LIN {X 0,Y 308.465,Z 992.055,A -85,B 0,C 180,E1 8309.518,E2 8309.518} C_VEL
LIN {X 0,Y 302.888,Z 996.087,A -85,B 0,C 180,E1 8308.383,E2 8308.383} C_VEL
LIN {X 0,Y 297.097,Z 1000.732,A -85,B 0,C 180,E1 8307.239,E2 8307.239} C_VEL
LIN {X 0,Y 292.705,Z 1003.413,A -85,B 0,C 180,E1 8306.146,E2 8306.146} C_VEL
LIN {X 0,Y 288.012,Z 1006.83,A -85,B 0,C 180,E1 8305.058,E2 8305.058} C_VEL
LIN {X 0,Y 284.129,Z 1009.021,A -85,B 0,C 180,E1 8303.872,E2 8303.872} C_VEL
LIN {X 0,Y 279.973,Z 1011.868,A -85,B 0,C 180,E1 8302.688,E2 8302.688} C_VEL
LIN {X 0,Y 277.713,Z 1012.755,A -85,B 0,C 180,E1 8301.768,E2 8301.768} C_VEL
LIN {X 0,Y 274.229,Z 1015.152,A -85,B 0,C 180,E1 8300.712,E2 8300.712} C_VEL
LIN {X 0,Y 271.961,Z 1016.233,A -85,B 0,C 180,E1 8299.546,E2 8299.546} C_VEL
LIN {X 0,Y 271.367,Z 1019.443,A -85,B 0,C 180,E1 8298.697,E2 8298.697} C_VEL
LIN {X 0,Y 269.802,Z 1031.042,A -85,B 0,C 180,E1 8295.696,E2 8295.696} C_VEL
LIN {X 0,Y 268.586,Z 1041.049,A -85,B 0,C 180,E1 8292.47,E2 8292.47} C_VEL
LIN {X 0,Y 267.824,Z 1048.97,A -85,B 0,C 180,E1 8289.238,E2 8289.238} C_VEL
LIN {X 0,Y 267.45,Z 1055.351,A -85,B 0,C 180,E1 8285.794,E2 8285.794} C_VEL
LIN {X 0,Y 267.481,Z 1059.896,A -85,B 0,C 180,E1 8282.357,E2 8282.357} C_VEL
LIN {X 0,Y 267.867,Z 1062.688,A -85,B 0,C 180,E1 8278.931,E2 8278.931} C_VEL
LIN {X 0,Y 268.592,Z 1063.764,A -85,B 0,C 180,E1 8275.517,E2 8275.517} C_VEL
LIN {X 0,Y 269.756,Z 1063.163,A -85,B 0,C 180,E1 8272.118,E2 8272.118} C_VEL
LIN {X 0,Y 271.423,Z 1060.847,A -85,B 0,C 180,E1 8268.742,E2 8268.742} C_VEL
LIN {X 0,Y 273.467,Z 1056.96,A -85,B 0,C 180,E1 8265.605,E2 8265.605} C_VEL
LIN {X 0,Y 276.201,Z 1050.914,A -85,B 0,C 180,E1 8262.298,E2 8262.298} C_VEL
LIN {X 0,Y 279.28,Z 1043.229,A -85,B 0,C 180,E1 8259.242,E2 8259.242} C_VEL
LIN {X 0,Y 282.707,Z 1033.633,A -85,B 0,C 180,E1 8256.351,E2 8256.351} C_VEL
LIN {X 0,Y 285.415,Z 1026.001,A -85,B 0,C 180,E1 8254.421,E2 8254.421} C_VEL
LIN {X 0,Y 288.972,Z 1024.505,A -85,B 0,C 180,E1 8253.491,E2 8253.491} C_VEL
LIN {X 0,Y 291.755,Z 1023.074,A -85,B 0,C 180,E1 8252.884,E2 8252.884} C_VEL
LIN {X 0,Y 296.745,Z 1020.577,A -85,B 0,C 180,E1 8251.855,E2 8251.855} C_VEL
LIN {X 0,Y 303.495,Z 1016.999,A -85,B 0,C 180,E1 8250.602,E2 8250.602} C_VEL
LIN {X 0,Y 312.335,Z 1011.631,A -85,B 0,C 180,E1 8249.19,E2 8249.19} C_VEL
LIN {X 0,Y 321.708,Z 1005.383,A -85,B 0,C 180,E1 8247.896,E2 8247.896} C_VEL
LIN {X 0,Y 326.811,Z 1001.618,A -85,B 0,C 180,E1 8247.283,E2 8247.283} C_VEL
LIN {X 0,Y 332.766,Z 996.983,A -85,B 0,C 180,E1 8246.592,E2 8246.592} C_VEL
LIN {X 0,Y 325.704,Z 1016.942,A -85,B 0,C 180,E1 8244.744,E2 8244.744} C_VEL
LIN {X 0,Y 318.629,Z 1034.815,A -85,B 0,C 180,E1 8242.726,E2 8242.726} C_VEL
LIN {X 0,Y 310.317,Z 1054.234,A -85,B 0,C 180,E1 8240.072,E2 8240.072} C_VEL
LIN {X 0,Y 302.689,Z 1070.961,A -85,B 0,C 180,E1 8237.305,E2 8237.305} C_VEL
LIN {X 0,Y 294.934,Z 1087.108,A -85,B 0,C 180,E1 8234.053,E2 8234.053} C_VEL
LIN {X 0,Y 287.656,Z 1102.055,A -85,B 0,C 180,E1 8230.429,E2 8230.429} C_VEL
LIN {X 0,Y 281.386,Z 1114.908,A -85,B 0,C 180,E1 8226.653,E2 8226.653} C_VEL
LIN {X 0,Y 275.565,Z 1127.286,A -85,B 0,C 180,E1 8222.234,E2 8222.234} C_VEL
LIN {X 0,Y 271.069,Z 1137.736,A -85,B 0,C 180,E1 8217.695,E2 8217.695} C_VEL
LIN {X 0,Y 267.812,Z 1146.209,A -85,B 0,C 180,E1 8213.08,E2 8213.08} C_VEL
LIN {X 0,Y 265.626,Z 1153.374,A -85,B 0,C 180,E1 8208.206,E2 8208.206} C_VEL
LIN {X 0,Y 264.507,Z 1158.372,A -85,B 0,C 180,E1 8203.719,E2 8203.719} C_VEL
LIN {X 0,Y 264.05,Z 1162.21,A -85,B 0,C 180,E1 8198.931,E2 8198.931} C_VEL
LIN {X 0,Y 263.973,Z 1164.181,A -85,B 0,C 180,E1 8194.78,E2 8194.78} C_VEL
LIN {X 0,Y 263.978,Z 1164.983,A -85,B 0,C 180,E1 8190.868,E2 8190.868} C_VEL
LIN {X 0,Y 263.962,Z 1164.612,A -85,B 0,C 180,E1 8186.525,E2 8186.525} C_VEL
LIN {X 0,Y 263.986,Z 1162.932,A -85,B 0,C 180,E1 8182.382,E2 8182.382} C_VEL
LIN {X 0,Y 264.232,Z 1160.273,A -85,B 0,C 180,E1 8178.431,E2 8178.431} C_VEL
LIN {X 0,Y 265.089,Z 1155.51,A -85,B 0,C 180,E1 8173.568,E2 8173.568} C_VEL
LIN {X 0,Y 266.681,Z 1149.663,A -85,B 0,C 180,E1 8169.134,E2 8169.134} C_VEL
LIN {X 0,Y 269.694,Z 1141.104,A -85,B 0,C 180,E1 8164.057,E2 8164.057} C_VEL
LIN {X 0,Y 273.705,Z 1131.511,A -85,B 0,C 180,E1 8159.484,E2 8159.484} C_VEL
LIN {X 0,Y 278.726,Z 1120.423,A -85,B 0,C 180,E1 8155.224,E2 8155.224} C_VEL
LIN {X 0,Y 284.969,Z 1107.485,A -85,B 0,C 180,E1 8151.093,E2 8151.093} C_VEL
LIN {X 0,Y 291.692,Z 1093.705,A -85,B 0,C 180,E1 8147.473,E2 8147.473} C_VEL
LIN {X 0,Y 299.455,Z 1077.629,A -85,B 0,C 180,E1 8143.986,E2 8143.986} C_VEL
LIN {X 0,Y 307.272,Z 1060.949,A -85,B 0,C 180,E1 8140.981,E2 8140.981} C_VEL
LIN {X 0,Y 315.017,Z 1043.264,A -85,B 0,C 180,E1 8138.374,E2 8138.374} C_VEL
LIN {X 0,Y 323.045,Z 1023.596,A -85,B 0,C 180,E1 8135.98,E2 8135.98} C_VEL
LIN {X 0,Y 330.114,Z 1004.598,A -85,B 0,C 180,E1 8134.078,E2 8134.078} C_VEL
LIN {X 0,Y 336.583,Z 984.934,A -85,B 0,C 180,E1 8132.472,E2 8132.472} C_VEL
LIN {X 0,Y 342.744,Z 963.75,A -85,B 0,C 180,E1 8131.059,E2 8131.059} C_VEL
LIN {X 0,Y 347.877,Z 942.3,A -85,B 0,C 180,E1 8129.938,E2 8129.938} C_VEL
LIN {X 0,Y 352.415,Z 919.016,A -85,B 0,C 180,E1 8129.004,E2 8129.004} C_VEL
LIN {X 0,Y 355.597,Z 897.104,A -85,B 0,C 180,E1 8128.357,E2 8128.357} C_VEL
LIN {X 0,Y 358.517,Z 862.586,A -85,B 0,C 180,E1 8127.602,E2 8127.602} C_VEL
LIN {X 0,Y 372.306,Z 678.191,A -85,B 0,C 180,E1 8123.839,E2 8123.839} C_VEL
LIN {X 0,Y 365.076,Z 666.2,A -85,B 0,C 180,E1 8120.857,E2 8120.857} C_VEL
LIN {X 0,Y 358.906,Z 656.732,A -85,B 0,C 180,E1 8117.928,E2 8117.928} C_VEL
LIN {X 0,Y 354.027,Z 649.555,A -85,B 0,C 180,E1 8115.227,E2 8115.227} C_VEL
LIN {X 0,Y 350.238,Z 644.346,A -85,B 0,C 180,E1 8112.782,E2 8112.782} C_VEL
LIN {X 0,Y 347.182,Z 640.185,A -85,B 0,C 180,E1 8110.453,E2 8110.453} C_VEL
LIN {X 0,Y 343.492,Z 635.283,A -85,B 0,C 180,E1 8106.854,E2 8106.854} C_VEL
LIN {X 0,Y 339.862,Z 631.157,A -85,B 0,C 180,E1 8100.505,E2 8100.505} C_VEL
LIN {X 0,Y 339.408,Z 630.8,A -85,B 0,C 180,E1 8097.467,E2 8097.467} C_VEL
LIN {X 0,Y 339.995,Z 632.727,A -85,B 0,C 180,E1 8093.414,E2 8093.414} C_VEL
LIN {X 0,Y 341.873,Z 635.288,A -85,B 0,C 180,E1 8089.808,E2 8089.808} C_VEL
LIN {X 0,Y 345.158,Z 640.526,A -85,B 0,C 180,E1 8085.916,E2 8085.916} C_VEL
LIN {X 0,Y 348.455,Z 645.83,A -85,B 0,C 180,E1 8083.067,E2 8083.067} C_VEL
LIN {X 0,Y 351.262,Z 650.243,A -85,B 0,C 180,E1 8081.064,E2 8081.064} C_VEL
LIN {X 0,Y 355.585,Z 657.064,A -85,B 0,C 180,E1 8078.429,E2 8078.429} C_VEL
LIN {X 0,Y 361.502,Z 667.073,A -85,B 0,C 180,E1 8075.357,E2 8075.357} C_VEL
LIN {X 0,Y 367.869,Z 678.378,A -85,B 0,C 180,E1 8072.524,E2 8072.524} C_VEL
LIN {X 0,Y 370.099,Z 682.724,A -85,B 0,C 180,E1 8071.607,E2 8071.607} C_VEL
LIN {X 0,Y 355.361,Z 895.308,A -85,B 0,C 180,E1 8067.466,E2 8067.466} C_VEL
LIN {X 0,Y 352.442,Z 917.469,A -85,B 0,C 180,E1 8066.87,E2 8066.87} C_VEL
LIN {X 0,Y 348.535,Z 938.899,A -85,B 0,C 180,E1 8066.077,E2 8066.077} C_VEL
LIN {X 0,Y 344.048,Z 958.089,A -85,B 0,C 180,E1 8065.133,E2 8065.133} C_VEL
LIN {X 0,Y 338.162,Z 979.093,A -85,B 0,C 180,E1 8063.823,E2 8063.823} C_VEL
LIN {X 0,Y 332.048,Z 997.764,A -85,B 0,C 180,E1 8062.368,E2 8062.368} C_VEL
LIN {X 0,Y 324.986,Z 1016.544,A -85,B 0,C 180,E1 8060.555,E2 8060.555} C_VEL
LIN {X 0,Y 317.727,Z 1034.044,A -85,B 0,C 180,E1 8058.501,E2 8058.501} C_VEL
LIN {X 0,Y 310.143,Z 1050.573,A -85,B 0,C 180,E1 8056.121,E2 8056.121} C_VEL
LIN {X 0,Y 302.083,Z 1066.923,A -85,B 0,C 180,E1 8053.247,E2 8053.247} C_VEL
LIN {X 0,Y 294.604,Z 1081.378,A -85,B 0,C 180,E1 8050.154,E2 8050.154} C_VEL
LIN {X 0,Y 287.561,Z 1094.347,A -85,B 0,C 180,E1 8046.731,E2 8046.731} C_VEL
LIN {X 0,Y 280.871,Z 1106.615,A -85,B 0,C 180,E1 8042.758,E2 8042.758} C_VEL
LIN {X 0,Y 275.408,Z 1116.941,A -85,B 0,C 180,E1 8038.635,E2 8038.635} C_VEL
LIN {X 0,Y 270.941,Z 1125.73,A -85,B 0,C 180,E1 8034.181,E2 8034.181} C_VEL
LIN {X 0,Y 267.62,Z 1133.095,A -85,B 0,C 180,E1 8029.421,E2 8029.421} C_VEL
LIN {X 0,Y 265.617,Z 1138.539,A -85,B 0,C 180,E1 8024.831,E2 8024.831} C_VEL
LIN {X 0,Y 264.545,Z 1142.323,A -85,B 0,C 180,E1 8020.232,E2 8020.232} C_VEL
LIN {X 0,Y 264.103,Z 1144.788,A -85,B 0,C 180,E1 8015.649,E2 8015.649} C_VEL
LIN {X 0,Y 264.011,Z 1145.742,A -85,B 0,C 180,E1 8011.302,E2 8011.302} C_VEL
LIN {X 0,Y 264.024,Z 1145.579,A -85,B 0,C 180,E1 8006.961,E2 8006.961} C_VEL
LIN {X 0,Y 264.22,Z 1143.987,A -85,B 0,C 180,E1 8002.509,E2 8002.509} C_VEL
LIN {X 0,Y 264.879,Z 1141.055,A -85,B 0,C 180,E1 7997.87,E2 7997.87} C_VEL
LIN {X 0,Y 266.314,Z 1136.484,A -85,B 0,C 180,E1 7993.196,E2 7993.196} C_VEL
LIN {X 0,Y 269.053,Z 1129.799,A -85,B 0,C 180,E1 7988.184,E2 7988.184} C_VEL
LIN {X 0,Y 272.827,Z 1121.996,A -85,B 0,C 180,E1 7983.676,E2 7983.676} C_VEL
LIN {X 0,Y 277.801,Z 1112.388,A -85,B 0,C 180,E1 7979.341,E2 7979.341} C_VEL
LIN {X 0,Y 283.954,Z 1101.024,A -85,B 0,C 180,E1 7975.219,E2 7975.219} C_VEL
LIN {X 0,Y 290.839,Z 1088.462,A -85,B 0,C 180,E1 7971.519,E2 7971.519} C_VEL
LIN {X 0,Y 297.873,Z 1075.192,A -85,B 0,C 180,E1 7968.347,E2 7968.347} C_VEL
LIN {X 0,Y 305.973,Z 1059.295,A -85,B 0,C 180,E1 7965.234,E2 7965.234} C_VEL
LIN {X 0,Y 310.204,Z 1050.584,A -85,B 0,C 180,E1 7963.776,E2 7963.776} C_VEL
LIN {X 0,Y 312.062,Z 1045.27,A -85,B 0,C 180,E1 7962.81,E2 7962.81} C_VEL
LIN {X 0,Y 314.292,Z 1031.888,A -85,B 0,C 180,E1 7960.095,E2 7960.095} C_VEL
LIN {X 0,Y 316.243,Z 1025.963,A -85,B 0,C 180,E1 7959.231,E2 7959.231} C_VEL
LIN {X 0,Y 324.268,Z 1006.326,A -85,B 0,C 180,E1 7957.149,E2 7957.149} C_VEL
LIN {X 0,Y 331.11,Z 987.486,A -85,B 0,C 180,E1 7955.529,E2 7955.529} C_VEL
LIN {X 0,Y 335.993,Z 971.645,A -85,B 0,C 180,E1 7954.403,E2 7954.403} C_VEL
LIN {X 0,Y 330.589,Z 977.083,A -85,B 0,C 180,E1 7953.722,E2 7953.722} C_VEL
LIN {X 0,Y 323.686,Z 984.266,A -85,B 0,C 180,E1 7952.934,E2 7952.934} C_VEL
LIN {X 0,Y 316.957,Z 990.052,A -85,B 0,C 180,E1 7951.942,E2 7951.942} C_VEL
LIN {X 0,Y 313.068,Z 993.358,A -85,B 0,C 180,E1 7951.372,E2 7951.372} C_VEL
LIN {X 0,Y 305.966,Z 999.179,A -85,B 0,C 180,E1 7950.216,E2 7950.216} C_VEL
LIN {X 0,Y 301.655,Z 1002.099,A -85,B 0,C 180,E1 7949.378,E2 7949.378} C_VEL
LIN {X 0,Y 295.641,Z 1006.57,A -85,B 0,C 180,E1 7948.261,E2 7948.261} C_VEL
LIN {X 0,Y 290.401,Z 1009.846,A -85,B 0,C 180,E1 7947.032,E2 7947.032} C_VEL
LIN {X 0,Y 285.061,Z 1013.4,A -85,B 0,C 180,E1 7945.782,E2 7945.782} C_VEL
LIN {X 0,Y 281.549,Z 1015.27,A -85,B 0,C 180,E1 7944.775,E2 7944.775} C_VEL
LIN {X 0,Y 276.925,Z 1018.136,A -85,B 0,C 180,E1 7943.495,E2 7943.495} C_VEL
LIN {X 0,Y 274.214,Z 1019.381,A -85,B 0,C 180,E1 7942.511,E2 7942.511} C_VEL
LIN {X 0,Y 270.333,Z 1021.776,A -85,B 0,C 180,E1 7941.252,E2 7941.252} C_VEL
LIN {X 0,Y 267.723,Z 1022.893,A -85,B 0,C 180,E1 7940.096,E2 7940.096} C_VEL
LIN {X 0,Y 264.674,Z 1024.759,A -85,B 0,C 180,E1 7938.959,E2 7938.959} C_VEL
LIN {X 0,Y 262.884,Z 1025.621,A -85,B 0,C 180,E1 7937.786,E2 7937.786} C_VEL
LIN {X 0,Y 261.135,Z 1038.389,A -85,B 0,C 180,E1 7933.959,E2 7933.959} C_VEL
LIN {X 0,Y 260.167,Z 1047.242,A -85,B 0,C 180,E1 7930.631,E2 7930.631} C_VEL
LIN {X 0,Y 259.621,Z 1054.468,A -85,B 0,C 180,E1 7927.08,E2 7927.08} C_VEL
LIN {X 0,Y 259.531,Z 1059.835,A -85,B 0,C 180,E1 7923.535,E2 7923.535} C_VEL
LIN {X 0,Y 259.82,Z 1063.351,A -85,B 0,C 180,E1 7920.001,E2 7920.001} C_VEL
LIN {X 0,Y 260.543,Z 1065.234,A -85,B 0,C 180,E1 7916.26,E2 7916.26} C_VEL
LIN {X 0,Y 261.684,Z 1065.286,A -85,B 0,C 180,E1 7912.757,E2 7912.757} C_VEL
LIN {X 0,Y 263.338,Z 1063.577,A -85,B 0,C 180,E1 7909.278,E2 7909.278} C_VEL
LIN {X 0,Y 265.727,Z 1059.828,A -85,B 0,C 180,E1 7905.621,E2 7905.621} C_VEL
LIN {X 0,Y 268.397,Z 1054.726,A -85,B 0,C 180,E1 7902.438,E2 7902.438} C_VEL
LIN {X 0,Y 271.579,Z 1047.72,A -85,B 0,C 180,E1 7899.303,E2 7899.303} C_VEL
LIN {X 0,Y 275.057,Z 1039.306,A -85,B 0,C 180,E1 7896.431,E2 7896.431} C_VEL
LIN {X 0,Y 277.235,Z 1034.271,A -85,B 0,C 180,E1 7894.928,E2 7894.928} C_VEL
LIN {X 0,Y 281.19,Z 1032.783,A -85,B 0,C 180,E1 7893.838,E2 7893.838} C_VEL
LIN {X 0,Y 287.246,Z 1030.196,A -85,B 0,C 180,E1 7892.423,E2 7892.423} C_VEL
LIN {X 0,Y 294.527,Z 1026.845,A -85,B 0,C 180,E1 7890.958,E2 7890.958} C_VEL
LIN {X 0,Y 302.933,Z 1022.356,A -85,B 0,C 180,E1 7889.481,E2 7889.481} C_VEL
LIN {X 0,Y 311.29,Z 1017.573,A -85,B 0,C 180,E1 7888.213,E2 7888.213} C_VEL
LIN {X 0,Y 321.765,Z 1010.786,A -85,B 0,C 180,E1 7886.846,E2 7886.846} C_VEL
LIN {X 0,Y 323.628,Z 1009.421,A -85,B 0,C 180,E1 7886.638,E2 7886.638} C_VEL
LIN {X 0,Y 315.936,Z 1029.029,A -85,B 0,C 180,E1 7884.58,E2 7884.58} C_VEL
LIN {X 0,Y 308.001,Z 1047.314,A -85,B 0,C 180,E1 7882.23,E2 7882.23} C_VEL
LIN {X 0,Y 299.535,Z 1065.454,A -85,B 0,C 180,E1 7879.39,E2 7879.39} C_VEL
LIN {X 0,Y 291.628,Z 1081.602,A -85,B 0,C 180,E1 7876.338,E2 7876.338} C_VEL
LIN {X 0,Y 283.839,Z 1096.749,A -85,B 0,C 180,E1 7872.834,E2 7872.834} C_VEL
LIN {X 0,Y 276.368,Z 1111.283,A -85,B 0,C 180,E1 7868.748,E2 7868.748} C_VEL
LIN {X 0,Y 270.14,Z 1123.702,A -85,B 0,C 180,E1 7864.492,E2 7864.492} C_VEL
LIN {X 0,Y 264.931,Z 1134.572,A -85,B 0,C 180,E1 7859.879,E2 7859.879} C_VEL
LIN {X 0,Y 260.916,Z 1144.044,A -85,B 0,C 180,E1 7854.932,E2 7854.932} C_VEL
LIN {X 0,Y 258.433,Z 1150.971,A -85,B 0,C 180,E1 7850.378,E2 7850.378} C_VEL
LIN {X 0,Y 256.814,Z 1156.919,A -85,B 0,C 180,E1 7845.352,E2 7845.352} C_VEL
LIN {X 0,Y 256.174,Z 1160.665,A -85,B 0,C 180,E1 7841.026,E2 7841.026} C_VEL
LIN {X 0,Y 255.982,Z 1163.366,A -85,B 0,C 180,E1 7836.504,E2 7836.504} C_VEL
LIN {X 0,Y 255.992,Z 1164.572,A -85,B 0,C 180,E1 7832.015,E2 7832.015} C_VEL
LIN {X 0,Y 255.993,Z 1164.595,A -85,B 0,C 180,E1 7828.209,E2 7828.209} C_VEL
LIN {X 0,Y 255.97,Z 1163.518,A -85,B 0,C 180,E1 7823.946,E2 7823.946} C_VEL
LIN {X 0,Y 256.127,Z 1160.994,A -85,B 0,C 180,E1 7819.428,E2 7819.428} C_VEL
LIN {X 0,Y 256.718,Z 1157.345,A -85,B 0,C 180,E1 7815.105,E2 7815.105} C_VEL
LIN {X 0,Y 258.237,Z 1151.588,A -85,B 0,C 180,E1 7810.079,E2 7810.079} C_VEL
LIN {X 0,Y 260.734,Z 1144.469,A -85,B 0,C 180,E1 7805.344,E2 7805.344} C_VEL
LIN {X 0,Y 264.764,Z 1134.908,A -85,B 0,C 180,E1 7800.292,E2 7800.292} C_VEL
LIN {X 0,Y 269.882,Z 1124.197,A -85,B 0,C 180,E1 7795.706,E2 7795.706} C_VEL
LIN {X 0,Y 276.016,Z 1111.888,A -85,B 0,C 180,E1 7791.46,E2 7791.46} C_VEL
LIN {X 0,Y 283.428,Z 1097.473,A -85,B 0,C 180,E1 7787.365,E2 7787.365} C_VEL
LIN {X 0,Y 290.827,Z 1083.025,A -85,B 0,C 180,E1 7783.984,E2 7783.984} C_VEL
LIN {X 0,Y 298.808,Z 1066.835,A -85,B 0,C 180,E1 7780.867,E2 7780.867} C_VEL
LIN {X 0,Y 306.909,Z 1049.674,A -85,B 0,C 180,E1 7778.115,E2 7778.115} C_VEL
LIN {X 0,Y 314.598,Z 1031.966,A -85,B 0,C 180,E1 7775.787,E2 7775.787} C_VEL
LIN {X 0,Y 322.793,Z 1011.438,A -85,B 0,C 180,E1 7773.567,E2 7773.567} C_VEL
LIN {X 0,Y 329.957,Z 991.415,A -85,B 0,C 180,E1 7771.805,E2 7771.805} C_VEL
LIN {X 0,Y 336.446,Z 970.408,A -85,B 0,C 180,E1 7770.326,E2 7770.326} C_VEL
LIN {X 0,Y 342.171,Z 948.852,A -85,B 0,C 180,E1 7769.107,E2 7769.107} C_VEL
LIN {X 0,Y 346.805,Z 927.205,A -85,B 0,C 180,E1 7768.161,E2 7768.161} C_VEL
LIN {X 0,Y 350.76,Z 903.276,A -85,B 0,C 180,E1 7767.394,E2 7767.394} C_VEL
LIN {X 0,Y 353.294,Z 879.798,A -85,B 0,C 180,E1 7766.833,E2 7766.833} C_VEL
LIN {X 0,Y 368.448,Z 682.805,A -85,B 0,C 180,E1 7762.812,E2 7762.812} C_VEL
LIN {X 0,Y 361.881,Z 671.774,A -85,B 0,C 180,E1 7759.951,E2 7759.951} C_VEL
LIN {X 0,Y 356.205,Z 662.826,A -85,B 0,C 180,E1 7757.099,E2 7757.099} C_VEL
LIN {X 0,Y 351.6,Z 656.045,A -85,B 0,C 180,E1 7754.408,E2 7754.408} C_VEL
LIN {X 0,Y 348.445,Z 651.582,A -85,B 0,C 180,E1 7752.259,E2 7752.259} C_VEL
LIN {X 0,Y 345.794,Z 647.871,A -85,B 0,C 180,E1 7750.159,E2 7750.159} C_VEL
LIN {X 0,Y 342.363,Z 643.155,A -85,B 0,C 180,E1 7746.708,E2 7746.708} C_VEL
LIN {X 0,Y 338.841,Z 639.045,A -85,B 0,C 180,E1 7740.338,E2 7740.338} C_VEL
LIN {X 0,Y 338.433,Z 638.746,A -85,B 0,C 180,E1 7737.46,E2 7737.46} C_VEL
LIN {X 0,Y 339.079,Z 640.829,A -85,B 0,C 180,E1 7733.226,E2 7733.226} C_VEL
LIN {X 0,Y 340.737,Z 643.111,A -85,B 0,C 180,E1 7730.03,E2 7730.03} C_VEL
LIN {X 0,Y 343.857,Z 648.243,A -85,B 0,C 180,E1 7726.205,E2 7726.205} C_VEL
LIN {X 0,Y 347.066,Z 653.562,A -85,B 0,C 180,E1 7723.342,E2 7723.342} C_VEL
LIN {X 0,Y 349.815,Z 658.024,A -85,B 0,C 180,E1 7721.329,E2 7721.329} C_VEL
LIN {X 0,Y 353.772,Z 664.454,A -85,B 0,C 180,E1 7718.842,E2 7718.842} C_VEL
LIN {X 0,Y 359.491,Z 674.372,A -85,B 0,C 180,E1 7715.779,E2 7715.779} C_VEL
LIN {X 0,Y 365.641,Z 685.618,A -85,B 0,C 180,E1 7712.959,E2 7712.959} C_VEL
LIN {X 0,Y 366.33,Z 687.354,A -85,B 0,C 180,E1 7712.647,E2 7712.647} C_VEL
LIN {X 0,Y 351.355,Z 895.604,A -85,B 0,C 180,E1 7708.589,E2 7708.589} C_VEL
LIN {X 0,Y 348.322,Z 917.825,A -85,B 0,C 180,E1 7707.991,E2 7707.991} C_VEL
LIN {X 0,Y 344.33,Z 939.046,A -85,B 0,C 180,E1 7707.209,E2 7707.209} C_VEL
LIN {X 0,Y 339.631,Z 958.56,A -85,B 0,C 180,E1 7706.252,E2 7706.252} C_VEL
LIN {X 0,Y 333.505,Z 979.699,A -85,B 0,C 180,E1 7704.931,E2 7704.931} C_VEL
LIN {X 0,Y 327.214,Z 998.316,A -85,B 0,C 180,E1 7703.48,E2 7703.48} C_VEL
LIN {X 0,Y 319.935,Z 1017.014,A -85,B 0,C 180,E1 7701.668,E2 7701.668} C_VEL
LIN {X 0,Y 312.275,Z 1034.784,A -85,B 0,C 180,E1 7699.567,E2 7699.567} C_VEL
LIN {X 0,Y 304.273,Z 1051.601,A -85,B 0,C 180,E1 7697.121,E2 7697.121} C_VEL
LIN {X 0,Y 296.085,Z 1067.512,A -85,B 0,C 180,E1 7694.282,E2 7694.282} C_VEL
LIN {X 0,Y 288.416,Z 1081.718,A -85,B 0,C 180,E1 7691.199,E2 7691.199} C_VEL
LIN {X 0,Y 281.047,Z 1094.68,A -85,B 0,C 180,E1 7687.728,E2 7687.728} C_VEL
LIN {X 0,Y 274.019,Z 1106.935,A -85,B 0,C 180,E1 7683.685,E2 7683.685} C_VEL
LIN {X 0,Y 268.244,Z 1117.252,A -85,B 0,C 180,E1 7679.474,E2 7679.474} C_VEL
LIN {X 0,Y 263.495,Z 1126.038,A -85,B 0,C 180,E1 7674.911,E2 7674.911} C_VEL
LIN {X 0,Y 259.939,Z 1133.397,A -85,B 0,C 180,E1 7670.02,E2 7670.02} C_VEL
LIN {X 0,Y 257.777,Z 1138.839,A -85,B 0,C 180,E1 7665.293,E2 7665.293} C_VEL
LIN {X 0,Y 256.598,Z 1142.619,A -85,B 0,C 180,E1 7660.553,E2 7660.553} C_VEL
LIN {X 0,Y 256.12,Z 1145.08,A -85,B 0,C 180,E1 7655.826,E2 7655.826} C_VEL
LIN {X 0,Y 256.014,Z 1146.011,A -85,B 0,C 180,E1 7651.567,E2 7651.567} C_VEL
LIN {X 0,Y 256.024,Z 1145.918,A -85,B 0,C 180,E1 7647.314,E2 7647.314} C_VEL
LIN {X 0,Y 256.223,Z 1144.434,A -85,B 0,C 180,E1 7642.601,E2 7642.601} C_VEL
LIN {X 0,Y 256.835,Z 1141.79,A -85,B 0,C 180,E1 7638.093,E2 7638.093} C_VEL
LIN {X 0,Y 258.339,Z 1137.265,A -85,B 0,C 180,E1 7633.125,E2 7633.125} C_VEL
LIN {X 0,Y 261.013,Z 1131.115,A -85,B 0,C 180,E1 7628.187,E2 7628.187} C_VEL
LIN {X 0,Y 264.847,Z 1123.5,A -85,B 0,C 180,E1 7623.546,E2 7623.546} C_VEL
LIN {X 0,Y 270.019,Z 1114.03,A -85,B 0,C 180,E1 7619.022,E2 7619.022} C_VEL
LIN {X 0,Y 276.233,Z 1103.191,A -85,B 0,C 180,E1 7614.864,E2 7614.864} C_VEL
LIN {X 0,Y 282.869,Z 1091.584,A -85,B 0,C 180,E1 7611.27,E2 7611.27} C_VEL
LIN {X 0,Y 290.474,Z 1078.009,A -85,B 0,C 180,E1 7607.838,E2 7607.838} C_VEL
LIN {X 0,Y 298.508,Z 1063.135,A -85,B 0,C 180,E1 7604.757,E2 7604.757} C_VEL
LIN {X 0,Y 306.418,Z 1047.36,A -85,B 0,C 180,E1 7602.114,E2 7602.114} C_VEL
LIN {X 0,Y 314.814,Z 1029.24,A -85,B 0,C 180,E1 7599.629,E2 7599.629} C_VEL
LIN {X 0,Y 316.243,Z 1025.963,A -85,B 0,C 180,E1 7599.231,E2 7599.231} C_VEL
LIN {X 0,Y 318.225,Z 1020.054,A -85,B 0,C 180,E1 7598.394,E2 7598.394} C_VEL
LIN {X 0,Y 320.783,Z 1005.274,A -85,B 0,C 180,E1 7595.988,E2 7595.988} C_VEL
LIN {X 0,Y 322.594,Z 998.896,A -85,B 0,C 180,E1 7595.275,E2 7595.275} C_VEL
LIN {X 0,Y 326.776,Z 987.099,A -85,B 0,C 180,E1 7594.296,E2 7594.296} C_VEL
LIN {X 0,Y 318.788,Z 994.051,A -85,B 0,C 180,E1 7593.29,E2 7593.29} C_VEL
LIN {X 0,Y 313.89,Z 997.958,A -85,B 0,C 180,E1 7592.57,E2 7592.57} C_VEL
LIN {X 0,Y 306.366,Z 1003.945,A -85,B 0,C 180,E1 7591.479,E2 7591.479} C_VEL
LIN {X 0,Y 299.562,Z 1008.615,A -85,B 0,C 180,E1 7590.265,E2 7590.265} C_VEL
LIN {X 0,Y 292.835,Z 1013.248,A -85,B 0,C 180,E1 7589.003,E2 7589.003} C_VEL
LIN {X 0,Y 288.024,Z 1016.094,A -85,B 0,C 180,E1 7587.947,E2 7587.947} C_VEL
LIN {X 0,Y 281.961,Z 1019.795,A -85,B 0,C 180,E1 7586.54,E2 7586.54} C_VEL
LIN {X 0,Y 278.95,Z 1021.394,A -85,B 0,C 180,E1 7585.704,E2 7585.704} C_VEL
LIN {X 0,Y 273.98,Z 1024.322,A -85,B 0,C 180,E1 7584.355,E2 7584.355} C_VEL
LIN {X 0,Y 270.732,Z 1025.831,A -85,B 0,C 180,E1 7583.277,E2 7583.277} C_VEL
LIN {X 0,Y 266.299,Z 1028.211,A -85,B 0,C 180,E1 7581.822,E2 7581.822} C_VEL
LIN {X 0,Y 263.979,Z 1029.196,A -85,B 0,C 180,E1 7580.858,E2 7580.858} C_VEL
LIN {X 0,Y 260.488,Z 1031.115,A -85,B 0,C 180,E1 7579.509,E2 7579.509} C_VEL
LIN {X 0,Y 258.622,Z 1031.734,A -85,B 0,C 180,E1 7578.483,E2 7578.483} C_VEL
LIN {X 0,Y 255.417,Z 1033.544,A -85,B 0,C 180,E1 7577.074,E2 7577.074} C_VEL
LIN {X 0,Y 253.98,Z 1034.217,A -85,B 0,C 180,E1 7575.912,E2 7575.912} C_VEL
LIN {X 0,Y 252.592,Z 1045.046,A -85,B 0,C 180,E1 7572.111,E2 7572.111} C_VEL
LIN {X 0,Y 251.846,Z 1053.216,A -85,B 0,C 180,E1 7568.448,E2 7568.448} C_VEL
LIN {X 0,Y 251.609,Z 1059.417,A -85,B 0,C 180,E1 7564.788,E2 7564.788} C_VEL
LIN {X 0,Y 251.793,Z 1063.683,A -85,B 0,C 180,E1 7561.138,E2 7561.138} C_VEL
LIN {X 0,Y 252.432,Z 1066.381,A -85,B 0,C 180,E1 7557.276,E2 7557.276} C_VEL
LIN {X 0,Y 253.508,Z 1067.185,A -85,B 0,C 180,E1 7553.66,E2 7553.66} C_VEL
LIN {X 0,Y 255.105,Z 1066.224,A -85,B 0,C 180,E1 7550.07,E2 7550.07} C_VEL
LIN {X 0,Y 257.318,Z 1063.568,A -85,B 0,C 180,E1 7546.519,E2 7546.519} C_VEL
LIN {X 0,Y 260.168,Z 1059.109,A -85,B 0,C 180,E1 7543.018,E2 7543.018} C_VEL
LIN {X 0,Y 263.627,Z 1052.577,A -85,B 0,C 180,E1 7539.579,E2 7539.579} C_VEL
LIN {X 0,Y 267.485,Z 1044.456,A -85,B 0,C 180,E1 7536.425,E2 7536.425} C_VEL
LIN {X 0,Y 268.698,Z 1042.164,A -85,B 0,C 180,E1 7535.604,E2 7535.604} C_VEL
LIN {X 0,Y 272.87,Z 1040.758,A -85,B 0,C 180,E1 7534.344,E2 7534.344} C_VEL
LIN {X 0,Y 278.591,Z 1038.738,A -85,B 0,C 180,E1 7532.882,E2 7532.882} C_VEL
LIN {X 0,Y 285.56,Z 1035.832,A -85,B 0,C 180,E1 7531.335,E2 7531.335} C_VEL
LIN {X 0,Y 292.991,Z 1032.477,A -85,B 0,C 180,E1 7529.891,E2 7529.891} C_VEL
LIN {X 0,Y 301.371,Z 1028.331,A -85,B 0,C 180,E1 7528.502,E2 7528.502} C_VEL
LIN {X 0,Y 311.108,Z 1022.839,A -85,B 0,C 180,E1 7527.103,E2 7527.103} C_VEL
LIN {X 0,Y 314.414,Z 1020.841,A -85,B 0,C 180,E1 7526.678,E2 7526.678} C_VEL
LIN {X 0,Y 306.51,Z 1039.334,A -85,B 0,C 180,E1 7524.505,E2 7524.505} C_VEL
LIN {X 0,Y 298.235,Z 1056.835,A -85,B 0,C 180,E1 7521.986,E2 7521.986} C_VEL
LIN {X 0,Y 289.319,Z 1074.577,A -85,B 0,C 180,E1 7518.885,E2 7518.885} C_VEL
LIN {X 0,Y 281.01,Z 1090.43,A -85,B 0,C 180,E1 7515.498,E2 7515.498} C_VEL
LIN {X 0,Y 273.115,Z 1104.93,A -85,B 0,C 180,E1 7511.684,E2 7511.684} C_VEL
LIN {X 0,Y 266.072,Z 1118.018,A -85,B 0,C 180,E1 7507.501,E2 7507.501} C_VEL
LIN {X 0,Y 260.2,Z 1129.246,A -85,B 0,C 180,E1 7503.104,E2 7503.104} C_VEL
LIN {X 0,Y 255.285,Z 1139.36,A -85,B 0,C 180,E1 7498.209,E2 7498.209} C_VEL
LIN {X 0,Y 251.887,Z 1147.439,A -85,B 0,C 180,E1 7493.388,E2 7493.388} C_VEL
LIN {X 0,Y 249.632,Z 1153.97,A -85,B 0,C 180,E1 7488.332,E2 7488.332} C_VEL
LIN {X 0,Y 248.43,Z 1159.005,A -85,B 0,C 180,E1 7483.262,E2 7483.262} C_VEL
LIN {X 0,Y 248.033,Z 1162.23,A -85,B 0,C 180,E1 7478.344,E2 7478.344} C_VEL
LIN {X 0,Y 247.978,Z 1163.961,A -85,B 0,C 180,E1 7473.93,E2 7473.93} C_VEL
LIN {X 0,Y 247.99,Z 1164.448,A -85,B 0,C 180,E1 7469.538,E2 7469.538} C_VEL
LIN {X 0,Y 247.98,Z 1163.739,A -85,B 0,C 180,E1 7465.375,E2 7465.375} C_VEL
LIN {X 0,Y 248.047,Z 1161.979,A -85,B 0,C 180,E1 7461.189,E2 7461.189} C_VEL
LIN {X 0,Y 248.537,Z 1158.358,A -85,B 0,C 180,E1 7456.032,E2 7456.032} C_VEL
LIN {X 0,Y 249.744,Z 1153.556,A -85,B 0,C 180,E1 7451.32,E2 7451.32} C_VEL
LIN {X 0,Y 252.162,Z 1146.671,A -85,B 0,C 180,E1 7446.144,E2 7446.144} C_VEL
LIN {X 0,Y 255.546,Z 1138.772,A -85,B 0,C 180,E1 7441.488,E2 7441.488} C_VEL
LIN {X 0,Y 260.693,Z 1128.205,A -85,B 0,C 180,E1 7436.475,E2 7436.475} C_VEL
LIN {X 0,Y 266.724,Z 1116.781,A -85,B 0,C 180,E1 7432.064,E2 7432.064} C_VEL
LIN {X 0,Y 273.641,Z 1103.891,A -85,B 0,C 180,E1 7428.036,E2 7428.036} C_VEL
LIN {X 0,Y 281.687,Z 1088.999,A -85,B 0,C 180,E1 7424.192,E2 7424.192} C_VEL
LIN {X 0,Y 289.812,Z 1073.532,A -85,B 0,C 180,E1 7420.926,E2 7420.926} C_VEL
LIN {X 0,Y 298.448,Z 1056.246,A -85,B 0,C 180,E1 7417.938,E2 7417.938} C_VEL
LIN {X 0,Y 306.739,Z 1038.646,A -85,B 0,C 180,E1 7415.421,E2 7415.421} C_VEL
LIN {X 0,Y 314.867,Z 1019.555,A -85,B 0,C 180,E1 7413.202,E2 7413.202} C_VEL
LIN {X 0,Y 323.109,Z 998.069,A -85,B 0,C 180,E1 7411.171,E2 7411.171} C_VEL
LIN {X 0,Y 330.062,Z 977.575,A -85,B 0,C 180,E1 7409.609,E2 7409.609} C_VEL
LIN {X 0,Y 336.184,Z 956.083,A -85,B 0,C 180,E1 7408.315,E2 7408.315} C_VEL
LIN {X 0,Y 341.658,Z 932.954,A -85,B 0,C 180,E1 7407.227,E2 7407.227} C_VEL
LIN {X 0,Y 345.704,Z 911.251,A -85,B 0,C 180,E1 7406.466,E2 7406.466} C_VEL
LIN {X 0,Y 348.707,Z 887.805,A -85,B 0,C 180,E1 7405.861,E2 7405.861} C_VEL
LIN {X 0,Y 364.554,Z 689.512,A -85,B 0,C 180,E1 7401.812,E2 7401.812} C_VEL
LIN {X 0,Y 364.617,Z 687.297,A -85,B 0,C 180,E1 7401.727,E2 7401.727} C_VEL
LIN {X 0,Y 358.248,Z 676.429,A -85,B 0,C 180,E1 7398.763,E2 7398.763} C_VEL
LIN {X 0,Y 352.499,Z 667.366,A -85,B 0,C 180,E1 7395.632,E2 7395.632} C_VEL
LIN {X 0,Y 347.775,Z 660.269,A -85,B 0,C 180,E1 7392.536,E2 7392.536} C_VEL
LIN {X 0,Y 344.417,Z 655.556,A -85,B 0,C 180,E1 7389.862,E2 7389.862} C_VEL
LIN {X 0,Y 341.097,Z 650.894,A -85,B 0,C 180,E1 7386.395,E2 7386.395} C_VEL
LIN {X 0,Y 337.823,Z 646.934,A -85,B 0,C 180,E1 7380.169,E2 7380.169} C_VEL
LIN {X 0,Y 337.455,Z 646.727,A -85,B 0,C 180,E1 7377.282,E2 7377.282} C_VEL
LIN {X 0,Y 338.377,Z 649.277,A -85,B 0,C 180,E1 7372.529,E2 7372.529} C_VEL
LIN {X 0,Y 339.654,Z 651.054,A -85,B 0,C 180,E1 7370.169,E2 7370.169} C_VEL
LIN {X 0,Y 342.562,Z 655.958,A -85,B 0,C 180,E1 7366.496,E2 7366.496} C_VEL
LIN {X 0,Y 345.686,Z 661.292,A -85,B 0,C 180,E1 7363.619,E2 7363.619} C_VEL
LIN {X 0,Y 348.258,Z 665.598,A -85,B 0,C 180,E1 7361.676,E2 7361.676} C_VEL
LIN {X 0,Y 352,Z 671.884,A -85,B 0,C 180,E1 7359.246,E2 7359.246} C_VEL
LIN {X 0,Y 357.657,Z 681.929,A -85,B 0,C 180,E1 7356.13,E2 7356.13} C_VEL
LIN {X 0,Y 362.706,Z 691.656,A -85,B 0,C 180,E1 7353.714,E2 7353.714} C_VEL
LIN {X 0,Y 347.518,Z 895.563,A -85,B 0,C 180,E1 7349.745,E2 7349.745} C_VEL
LIN {X 0,Y 344.4,Z 917.803,A -85,B 0,C 180,E1 7349.15,E2 7349.15} C_VEL
LIN {X 0,Y 340.262,Z 939.193,A -85,B 0,C 180,E1 7348.368,E2 7348.368} C_VEL
LIN {X 0,Y 335.344,Z 959.043,A -85,B 0,C 180,E1 7347.4,E2 7347.4} C_VEL
LIN {X 0,Y 328.976,Z 980.302,A -85,B 0,C 180,E1 7346.071,E2 7346.071} C_VEL
LIN {X 0,Y 322.19,Z 999.733,A -85,B 0,C 180,E1 7344.55,E2 7344.55} C_VEL
LIN {X 0,Y 314.673,Z 1018.27,A -85,B 0,C 180,E1 7342.732,E2 7342.732} C_VEL
LIN {X 0,Y 306.074,Z 1037.295,A -85,B 0,C 180,E1 7340.43,E2 7340.43} C_VEL
LIN {X 0,Y 297.739,Z 1054.15,A -85,B 0,C 180,E1 7337.916,E2 7337.916} C_VEL
LIN {X 0,Y 289.444,Z 1069.456,A -85,B 0,C 180,E1 7335.085,E2 7335.085} C_VEL
LIN {X 0,Y 280.966,Z 1084.306,A -85,B 0,C 180,E1 7331.718,E2 7331.718} C_VEL
LIN {X 0,Y 273.445,Z 1097.055,A -85,B 0,C 180,E1 7328.167,E2 7328.167} C_VEL
LIN {X 0,Y 266.57,Z 1108.363,A -85,B 0,C 180,E1 7324.238,E2 7324.238} C_VEL
LIN {X 0,Y 260.326,Z 1118.885,A -85,B 0,C 180,E1 7319.7,E2 7319.7} C_VEL
LIN {X 0,Y 255.492,Z 1127.512,A -85,B 0,C 180,E1 7315.002,E2 7315.002} C_VEL
LIN {X 0,Y 251.877,Z 1134.566,A -85,B 0,C 180,E1 7309.962,E2 7309.962} C_VEL
LIN {X 0,Y 249.547,Z 1140.122,A -85,B 0,C 180,E1 7304.621,E2 7304.621} C_VEL
LIN {X 0,Y 248.495,Z 1143.667,A -85,B 0,C 180,E1 7299.729,E2 7299.729} C_VEL
LIN {X 0,Y 248.083,Z 1145.688,A -85,B 0,C 180,E1 7294.855,E2 7294.855} C_VEL
LIN {X 0,Y 248.018,Z 1146.409,A -85,B 0,C 180,E1 7290.462,E2 7290.462} C_VEL
LIN {X 0,Y 248.064,Z 1145.91,A -85,B 0,C 180,E1 7285.839,E2 7285.839} C_VEL
LIN {X 0,Y 248.329,Z 1144.301,A -85,B 0,C 180,E1 7281.432,E2 7281.432} C_VEL
LIN {X 0,Y 249.258,Z 1140.996,A -85,B 0,C 180,E1 7276.31,E2 7276.31} C_VEL
LIN {X 0,Y 251.124,Z 1136.301,A -85,B 0,C 180,E1 7271.372,E2 7271.372} C_VEL
LIN {X 0,Y 254.289,Z 1129.729,A -85,B 0,C 180,E1 7266.355,E2 7266.355} C_VEL
LIN {X 0,Y 258.959,Z 1121.291,A -85,B 0,C 180,E1 7261.395,E2 7261.395} C_VEL
LIN {X 0,Y 264.545,Z 1111.857,A -85,B 0,C 180,E1 7257.026,E2 7257.026} C_VEL
LIN {X 0,Y 271.032,Z 1101.052,A -85,B 0,C 180,E1 7253.035,E2 7253.035} C_VEL
LIN {X 0,Y 278.647,Z 1088.387,A -85,B 0,C 180,E1 7249.227,E2 7249.227} C_VEL
LIN {X 0,Y 286.373,Z 1075.055,A -85,B 0,C 180,E1 7245.988,E2 7245.988} C_VEL
LIN {X 0,Y 294.922,Z 1059.539,A -85,B 0,C 180,E1 7242.921,E2 7242.921} C_VEL
LIN {X 0,Y 303.103,Z 1043.737,A -85,B 0,C 180,E1 7240.358,E2 7240.358} C_VEL
LIN {X 0,Y 311.204,Z 1026.386,A -85,B 0,C 180,E1 7238.079,E2 7238.079} C_VEL
LIN {X 0,Y 319.48,Z 1006.817,A -85,B 0,C 180,E1 7236,E2 7236} C_VEL
LIN {X 0,Y 322.594,Z 998.896,A -85,B 0,C 180,E1 7235.275,E2 7235.275} C_VEL
LIN {X 0,Y 322.388,Z 997.968,A -85,B 0,C 180,E1 7235.047,E2 7235.047} C_VEL
LIN {X 0,Y 320.677,Z 998.091,A -85,B 0,C 180,E1 7234.591,E2 7234.591} C_VEL
LIN {X 0,Y 317.5,Z 999.976,A -85,B 0,C 180,E1 7234.051,E2 7234.051} C_VEL
LIN {X 0,Y 307.008,Z 1008.567,A -85,B 0,C 180,E1 7232.752,E2 7232.752} C_VEL
LIN {X 0,Y 306.32,Z 1009.064,A -85,B 0,C 180,E1 7232.647,E2 7232.647} C_VEL
LIN {X 0,Y 298.265,Z 1014.392,A -85,B 0,C 180,E1 7231.306,E2 7231.306} C_VEL
LIN {X 0,Y 290.944,Z 1019.133,A -85,B 0,C 180,E1 7230,E2 7230} C_VEL
LIN {X 0,Y 286.41,Z 1021.747,A -85,B 0,C 180,E1 7229.029,E2 7229.029} C_VEL
LIN {X 0,Y 279.718,Z 1025.65,A -85,B 0,C 180,E1 7227.565,E2 7227.565} C_VEL
LIN {X 0,Y 275.569,Z 1027.799,A -85,B 0,C 180,E1 7226.506,E2 7226.506} C_VEL
LIN {X 0,Y 269.987,Z 1030.736,A -85,B 0,C 180,E1 7224.973,E2 7224.973} C_VEL
LIN {X 0,Y 267.163,Z 1032.089,A -85,B 0,C 180,E1 7224.076,E2 7224.076} C_VEL
LIN {X 0,Y 262.222,Z 1034.563,A -85,B 0,C 180,E1 7222.415,E2 7222.415} C_VEL
LIN {X 0,Y 260.239,Z 1035.412,A -85,B 0,C 180,E1 7221.645,E2 7221.645} C_VEL
LIN {X 0,Y 256.196,Z 1037.355,A -85,B 0,C 180,E1 7220.087,E2 7220.087} C_VEL
LIN {X 0,Y 254.097,Z 1038.146,A -85,B 0,C 180,E1 7219.063,E2 7219.063} C_VEL
LIN {X 0,Y 250.587,Z 1039.842,A -85,B 0,C 180,E1 7217.413,E2 7217.413} C_VEL
LIN {X 0,Y 249.26,Z 1040.227,A -85,B 0,C 180,E1 7216.522,E2 7216.522} C_VEL
LIN {X 0,Y 246.479,Z 1041.732,A -85,B 0,C 180,E1 7215.048,E2 7215.048} C_VEL
LIN {X 0,Y 245.182,Z 1042.286,A -85,B 0,C 180,E1 7213.802,E2 7213.802} C_VEL
LIN {X 0,Y 244.06,Z 1052.562,A -85,B 0,C 180,E1 7209.432,E2 7209.432} C_VEL
LIN {X 0,Y 243.697,Z 1059.31,A -85,B 0,C 180,E1 7205.652,E2 7205.652} C_VEL
LIN {X 0,Y 243.816,Z 1064.2,A -85,B 0,C 180,E1 7201.881,E2 7201.881} C_VEL
LIN {X 0,Y 244.378,Z 1067.359,A -85,B 0,C 180,E1 7198.125,E2 7198.125} C_VEL
LIN {X 0,Y 245.394,Z 1068.769,A -85,B 0,C 180,E1 7194.389,E2 7194.389} C_VEL
LIN {X 0,Y 247.093,Z 1068.435,A -85,B 0,C 180,E1 7190.451,E2 7190.451} C_VEL
LIN {X 0,Y 249.354,Z 1066.394,A -85,B 0,C 180,E1 7186.788,E2 7186.788} C_VEL
LIN {X 0,Y 252.272,Z 1062.501,A -85,B 0,C 180,E1 7183.183,E2 7183.183} C_VEL
LIN {X 0,Y 255.878,Z 1056.747,A -85,B 0,C 180,E1 7179.65,E2 7179.65} C_VEL
LIN {X 0,Y 260.153,Z 1049.471,A -85,B 0,C 180,E1 7176.321,E2 7176.321} C_VEL
LIN {X 0,Y 264.394,Z 1048.334,A -85,B 0,C 180,E1 7174.942,E2 7174.942} C_VEL
LIN {X 0,Y 269.942,Z 1046.617,A -85,B 0,C 180,E1 7173.374,E2 7173.374} C_VEL
LIN {X 0,Y 275.874,Z 1044.538,A -85,B 0,C 180,E1 7171.891,E2 7171.891} C_VEL
LIN {X 0,Y 283.065,Z 1041.736,A -85,B 0,C 180,E1 7170.363,E2 7170.363} C_VEL
LIN {X 0,Y 290.727,Z 1038.523,A -85,B 0,C 180,E1 7168.945,E2 7168.945} C_VEL
LIN {X 0,Y 300.518,Z 1033.711,A -85,B 0,C 180,E1 7167.386,E2 7167.386} C_VEL
LIN {X 0,Y 305.065,Z 1031.545,A -85,B 0,C 180,E1 7166.697,E2 7166.697} C_VEL
LIN {X 0,Y 296.347,Z 1050.184,A -85,B 0,C 180,E1 7164.237,E2 7164.237} C_VEL
LIN {X 0,Y 287.616,Z 1067.205,A -85,B 0,C 180,E1 7161.461,E2 7161.461} C_VEL
LIN {X 0,Y 278.329,Z 1084.377,A -85,B 0,C 180,E1 7158.041,E2 7158.041} C_VEL
LIN {X 0,Y 270.008,Z 1099.224,A -85,B 0,C 180,E1 7154.418,E2 7154.418} C_VEL
LIN {X 0,Y 262.334,Z 1112.587,A -85,B 0,C 180,E1 7150.387,E2 7150.387} C_VEL
LIN {X 0,Y 255.458,Z 1124.834,A -85,B 0,C 180,E1 7145.886,E2 7145.886} C_VEL
LIN {X 0,Y 250.054,Z 1134.891,A -85,B 0,C 180,E1 7141.32,E2 7141.32} C_VEL
LIN {X 0,Y 245.551,Z 1144.165,A -85,B 0,C 180,E1 7136.089,E2 7136.089} C_VEL
LIN {X 0,Y 242.644,Z 1151.313,A -85,B 0,C 180,E1 7131.008,E2 7131.008} C_VEL
LIN {X 0,Y 240.916,Z 1156.758,A -85,B 0,C 180,E1 7125.898,E2 7125.898} C_VEL
LIN {X 0,Y 240.196,Z 1160.412,A -85,B 0,C 180,E1 7121.283,E2 7121.283} C_VEL
LIN {X 0,Y 239.981,Z 1163.012,A -85,B 0,C 180,E1 7116.219,E2 7116.219} C_VEL
LIN {X 0,Y 240.002,Z 1164.015,A -85,B 0,C 180,E1 7111.91,E2 7111.91} C_VEL
LIN {X 0,Y 240.002,Z 1164.013,A -85,B 0,C 180,E1 7108.09,E2 7108.09} C_VEL
LIN {X 0,Y 239.987,Z 1162.933,A -85,B 0,C 180,E1 7103.541,E2 7103.541} C_VEL
LIN {X 0,Y 240.221,Z 1160.229,A -85,B 0,C 180,E1 7098.475,E2 7098.475} C_VEL
LIN {X 0,Y 240.974,Z 1156.523,A -85,B 0,C 180,E1 7093.859,E2 7093.859} C_VEL
LIN {X 0,Y 242.982,Z 1150.333,A -85,B 0,C 180,E1 7088.263,E2 7088.263} C_VEL
LIN {X 0,Y 246.08,Z 1143.022,A -85,B 0,C 180,E1 7083.191,E2 7083.191} C_VEL
LIN {X 0,Y 250.538,Z 1133.896,A -85,B 0,C 180,E1 7078.211,E2 7078.211} C_VEL
LIN {X 0,Y 256.35,Z 1123.208,A -85,B 0,C 180,E1 7073.462,E2 7073.462} C_VEL
LIN {X 0,Y 263.197,Z 1111.005,A -85,B 0,C 180,E1 7069.11,E2 7069.11} C_VEL
LIN {X 0,Y 271.314,Z 1096.763,A -85,B 0,C 180,E1 7064.962,E2 7064.962} C_VEL
LIN {X 0,Y 279.815,Z 1081.681,A -85,B 0,C 180,E1 7061.376,E2 7061.376} C_VEL
LIN {X 0,Y 288.412,Z 1065.532,A -85,B 0,C 180,E1 7058.258,E2 7058.258} C_VEL
LIN {X 0,Y 297.496,Z 1047.569,A -85,B 0,C 180,E1 7055.41,E2 7055.41} C_VEL
LIN {X 0,Y 305.867,Z 1029.601,A -85,B 0,C 180,E1 7053.086,E2 7053.086} C_VEL
LIN {X 0,Y 313.966,Z 1010.398,A -85,B 0,C 180,E1 7051.056,E2 7051.056} C_VEL
LIN {X 0,Y 321.635,Z 990.188,A -85,B 0,C 180,E1 7049.31,E2 7049.31} C_VEL
LIN {X 0,Y 328.165,Z 970.063,A -85,B 0,C 180,E1 7047.923,E2 7047.923} C_VEL
LIN {X 0,Y 334.349,Z 947.816,A -85,B 0,C 180,E1 7046.696,E2 7046.696} C_VEL
LIN {X 0,Y 339.139,Z 926.463,A -85,B 0,C 180,E1 7045.788,E2 7045.788} C_VEL
LIN {X 0,Y 343.162,Z 903.023,A -85,B 0,C 180,E1 7045.058,E2 7045.058} C_VEL
LIN {X 0,Y 345.813,Z 879.399,A -85,B 0,C 180,E1 7044.5,E2 7044.5} C_VEL
LIN {X 0,Y 361.075,Z 692.134,A -85,B 0,C 180,E1 7040.695,E2 7040.695} C_VEL
LIN {X 0,Y 355.12,Z 681.873,A -85,B 0,C 180,E1 7037.745,E2 7037.745} C_VEL
LIN {X 0,Y 350.304,Z 674.109,A -85,B 0,C 180,E1 7034.969,E2 7034.969} C_VEL
LIN {X 0,Y 345.78,Z 667.233,A -85,B 0,C 180,E1 7031.847,E2 7031.847} C_VEL
LIN {X 0,Y 343.056,Z 663.241,A -85,B 0,C 180,E1 7029.562,E2 7029.562} C_VEL
LIN {X 0,Y 339.961,Z 658.751,A -85,B 0,C 180,E1 7026.229,E2 7026.229} C_VEL
LIN {X 0,Y 336.805,Z 654.824,A -85,B 0,C 180,E1 7020,E2 7020} C_VEL
LIN {X 0,Y 336.48,Z 654.677,A -85,B 0,C 180,E1 7017.274,E2 7017.274} C_VEL
LIN {X 0,Y 337.729,Z 657.687,A -85,B 0,C 180,E1 7011.83,E2 7011.83} C_VEL
LIN {X 0,Y 338.574,Z 658.995,A -85,B 0,C 180,E1 7010.309,E2 7010.309} C_VEL
LIN {X 0,Y 341.272,Z 663.671,A -85,B 0,C 180,E1 7006.789,E2 7006.789} C_VEL
LIN {X 0,Y 344.219,Z 668.85,A -85,B 0,C 180,E1 7003.981,E2 7003.981} C_VEL
LIN {X 0,Y 346.936,Z 673.557,A -85,B 0,C 180,E1 7001.865,E2 7001.865} C_VEL
LIN {X 0,Y 350.428,Z 679.657,A -85,B 0,C 180,E1 6999.541,E2 6999.541} C_VEL
LIN {X 0,Y 355.682,Z 689.275,A -85,B 0,C 180,E1 6996.561,E2 6996.561} C_VEL
LIN {X 0,Y 359.183,Z 696.289,A -85,B 0,C 180,E1 6994.796,E2 6994.796} C_VEL
LIN {X 0,Y 343.83,Z 895.447,A -85,B 0,C 180,E1 6990.927,E2 6990.927} C_VEL
LIN {X 0,Y 340.63,Z 917.739,A -85,B 0,C 180,E1 6990.337,E2 6990.337} C_VEL
LIN {X 0,Y 336.337,Z 939.334,A -85,B 0,C 180,E1 6989.555,E2 6989.555} C_VEL
LIN {X 0,Y 331.427,Z 958.652,A -85,B 0,C 180,E1 6988.624,E2 6988.624} C_VEL
LIN {X 0,Y 324.92,Z 979.909,A -85,B 0,C 180,E1 6987.313,E2 6987.313} C_VEL
LIN {X 0,Y 317.93,Z 999.409,A -85,B 0,C 180,E1 6985.803,E2 6985.803} C_VEL
LIN {X 0,Y 310.21,Z 1017.945,A -85,B 0,C 180,E1 6984,E2 6984} C_VEL
LIN {X 0,Y 301.608,Z 1036.473,A -85,B 0,C 180,E1 6981.784,E2 6981.784} C_VEL
LIN {X 0,Y 293.216,Z 1052.902,A -85,B 0,C 180,E1 6979.359,E2 6979.359} C_VEL
LIN {X 0,Y 284.785,Z 1068.009,A -85,B 0,C 180,E1 6976.616,E2 6976.616} C_VEL
LIN {X 0,Y 276.344,Z 1082.393,A -85,B 0,C 180,E1 6973.429,E2 6973.429} C_VEL
LIN {X 0,Y 268.229,Z 1095.451,A -85,B 0,C 180,E1 6969.834,E2 6969.834} C_VEL
LIN {X 0,Y 260.546,Z 1107.573,A -85,B 0,C 180,E1 6965.684,E2 6965.684} C_VEL
LIN {X 0,Y 254.097,Z 1117.871,A -85,B 0,C 180,E1 6961.293,E2 6961.293} C_VEL
LIN {X 0,Y 248.736,Z 1126.654,A -85,B 0,C 180,E1 6956.5,E2 6956.5} C_VEL
LIN {X 0,Y 244.616,Z 1134.086,A -85,B 0,C 180,E1 6951.259,E2 6951.259} C_VEL
LIN {X 0,Y 242.05,Z 1139.638,A -85,B 0,C 180,E1 6946.067,E2 6946.067} C_VEL
LIN {X 0,Y 240.687,Z 1143.359,A -85,B 0,C 180,E1 6941.017,E2 6941.017} C_VEL
LIN {X 0,Y 240.143,Z 1145.726,A -85,B 0,C 180,E1 6935.975,E2 6935.975} C_VEL
LIN {X 0,Y 240.026,Z 1146.614,A -85,B 0,C 180,E1 6931.432,E2 6931.432} C_VEL
LIN {X 0,Y 240.042,Z 1146.479,A -85,B 0,C 180,E1 6926.896,E2 6926.896} C_VEL
LIN {X 0,Y 240.276,Z 1144.996,A -85,B 0,C 180,E1 6922.053,E2 6922.053} C_VEL
LIN {X 0,Y 241.079,Z 1142.237,A -85,B 0,C 180,E1 6917.073,E2 6917.073} C_VEL
LIN {X 0,Y 242.796,Z 1137.86,A -85,B 0,C 180,E1 6912.009,E2 6912.009} C_VEL
LIN {X 0,Y 245.911,Z 1131.715,A -85,B 0,C 180,E1 6906.767,E2 6906.767} C_VEL
LIN {X 0,Y 250.281,Z 1124.108,A -85,B 0,C 180,E1 6901.874,E2 6901.874} C_VEL
LIN {X 0,Y 256.099,Z 1114.652,A -85,B 0,C 180,E1 6897.133,E2 6897.133} C_VEL
LIN {X 0,Y 263.003,Z 1103.835,A -85,B 0,C 180,E1 6892.809,E2 6892.809} C_VEL
LIN {X 0,Y 270.304,Z 1092.235,A -85,B 0,C 180,E1 6889.101,E2 6889.101} C_VEL
LIN {X 0,Y 278.629,Z 1078.637,A -85,B 0,C 180,E1 6885.571,E2 6885.571} C_VEL
LIN {X 0,Y 287.297,Z 1063.861,A -85,B 0,C 180,E1 6882.455,E2 6882.455} C_VEL
LIN {X 0,Y 295.89,Z 1047.946,A -85,B 0,C 180,E1 6879.757,E2 6879.757} C_VEL
LIN {X 0,Y 305.069,Z 1029.439,A -85,B 0,C 180,E1 6877.209,E2 6877.209} C_VEL
LIN {X 0,Y 313.228,Z 1011.299,A -85,B 0,C 180,E1 6875.196,E2 6875.196} C_VEL
LIN {X 0,Y 317.551,Z 1000.459,A -85,B 0,C 180,E1 6874.166,E2 6874.166} C_VEL
LIN {X 0,Y 312.014,Z 1004.743,A -85,B 0,C 180,E1 6873.448,E2 6873.448} C_VEL
LIN {X 0,Y 306.32,Z 1009.064,A -85,B 0,C 180,E1 6872.647,E2 6872.647} C_VEL
LIN {X 0,Y 302.717,Z 1012.204,A -85,B 0,C 180,E1 6872.225,E2 6872.225} C_VEL
LIN {X 0,Y 293.397,Z 1021.846,A -85,B 0,C 180,E1 6871.636,E2 6871.636} C_VEL
LIN {X 0,Y 289.751,Z 1024.579,A -85,B 0,C 180,E1 6871.148,E2 6871.148} C_VEL
LIN {X 0,Y 283.185,Z 1028.211,A -85,B 0,C 180,E1 6869.858,E2 6869.858} C_VEL
LIN {X 0,Y 276.194,Z 1031.972,A -85,B 0,C 180,E1 6868.31,E2 6868.31} C_VEL
LIN {X 0,Y 267.083,Z 1036.571,A -85,B 0,C 180,E1 6865.977,E2 6865.977} C_VEL
LIN {X 0,Y 263.419,Z 1038.242,A -85,B 0,C 180,E1 6864.882,E2 6864.882} C_VEL
LIN {X 0,Y 257.93,Z 1040.693,A -85,B 0,C 180,E1 6863.05,E2 6863.05} C_VEL
LIN {X 0,Y 251.791,Z 1043.469,A -85,B 0,C 180,E1 6860.697,E2 6860.697} C_VEL
LIN {X 0,Y 249.491,Z 1044.417,A -85,B 0,C 180,E1 6859.645,E2 6859.645} C_VEL
LIN {X 0,Y 245.691,Z 1046.023,A -85,B 0,C 180,E1 6857.772,E2 6857.772} C_VEL
LIN {X 0,Y 244.121,Z 1046.649,A -85,B 0,C 180,E1 6856.906,E2 6856.906} C_VEL
LIN {X 0,Y 241.115,Z 1047.932,A -85,B 0,C 180,E1 6855.145,E2 6855.145} C_VEL
LIN {X 0,Y 239.964,Z 1048.272,A -85,B 0,C 180,E1 6854.232,E2 6854.232} C_VEL
LIN {X 0,Y 237.322,Z 1049.602,A -85,B 0,C 180,E1 6852.408,E2 6852.408} C_VEL
LIN {X 0,Y 236.458,Z 1050.212,A -85,B 0,C 180,E1 6851.161,E2 6851.161} C_VEL
LIN {X 0,Y 235.842,Z 1058.215,A -85,B 0,C 180,E1 6847.063,E2 6847.063} C_VEL
LIN {X 0,Y 235.809,Z 1063.922,A -85,B 0,C 180,E1 6843.16,E2 6843.16} C_VEL
LIN {X 0,Y 236.27,Z 1067.873,A -85,B 0,C 180,E1 6839.273,E2 6839.273} C_VEL
LIN {X 0,Y 237.193,Z 1070.055,A -85,B 0,C 180,E1 6835.407,E2 6835.407} C_VEL
LIN {X 0,Y 238.817,Z 1070.553,A -85,B 0,C 180,E1 6831.332,E2 6831.332} C_VEL
LIN {X 0,Y 241.032,Z 1069.319,A -85,B 0,C 180,E1 6827.544,E2 6827.544} C_VEL
LIN {X 0,Y 244.144,Z 1066.044,A -85,B 0,C 180,E1 6823.586,E2 6823.586} C_VEL
LIN {X 0,Y 247.841,Z 1061.129,A -85,B 0,C 180,E1 6819.946,E2 6819.946} C_VEL
LIN {X 0,Y 250.985,Z 1056.505,A -85,B 0,C 180,E1 6817.392,E2 6817.392} C_VEL
LIN {X 0,Y 255.454,Z 1055.511,A -85,B 0,C 180,E1 6815.735,E2 6815.735} C_VEL
LIN {X 0,Y 260.639,Z 1054.181,A -85,B 0,C 180,E1 6814.067,E2 6814.067} C_VEL
LIN {X 0,Y 271.013,Z 1051.119,A -85,B 0,C 180,E1 6811.341,E2 6811.341} C_VEL
LIN {X 0,Y 280.56,Z 1047.551,A -85,B 0,C 180,E1 6809.362,E2 6809.362} C_VEL
LIN {X 0,Y 289.615,Z 1043.759,A -85,B 0,C 180,E1 6807.762,E2 6807.762} C_VEL
LIN {X 0,Y 295.875,Z 1041.03,A -85,B 0,C 180,E1 6806.776,E2 6806.776} C_VEL
LIN {X 0,Y 287.535,Z 1057.46,A -85,B 0,C 180,E1 6804.372,E2 6804.372} C_VEL
LIN {X 0,Y 277.969,Z 1074.958,A -85,B 0,C 180,E1 6801.254,E2 6801.254} C_VEL
LIN {X 0,Y 269.286,Z 1090.103,A -85,B 0,C 180,E1 6797.954,E2 6797.954} C_VEL
LIN {X 0,Y 260.959,Z 1104,A -85,B 0,C 180,E1 6794.214,E2 6794.214} C_VEL
LIN {X 0,Y 253.239,Z 1116.873,A -85,B 0,C 180,E1 6790.008,E2 6790.008} C_VEL
LIN {X 0,Y 246.5,Z 1128.264,A -85,B 0,C 180,E1 6785.384,E2 6785.384} C_VEL
LIN {X 0,Y 240.759,Z 1138.601,A -85,B 0,C 180,E1 6780.166,E2 6780.166} C_VEL
LIN {X 0,Y 236.727,Z 1146.818,A -85,B 0,C 180,E1 6774.984,E2 6774.984} C_VEL
LIN {X 0,Y 234.065,Z 1153.236,A -85,B 0,C 180,E1 6769.723,E2 6769.723} C_VEL
LIN {X 0,Y 232.607,Z 1158.21,A -85,B 0,C 180,E1 6764.437,E2 6764.437} C_VEL
LIN {X 0,Y 232.064,Z 1161.52,A -85,B 0,C 180,E1 6759.173,E2 6759.173} C_VEL
LIN {X 0,Y 231.986,Z 1163.233,A -85,B 0,C 180,E1 6754.697,E2 6754.697} C_VEL
LIN {X 0,Y 232.013,Z 1163.908,A -85,B 0,C 180,E1 6750,E2 6750} C_VEL
LIN {X 0,Y 231.986,Z 1163.227,A -85,B 0,C 180,E1 6745.303,E2 6745.303} C_VEL
LIN {X 0,Y 232.064,Z 1161.51,A -85,B 0,C 180,E1 6740.827,E2 6740.827} C_VEL
LIN {X 0,Y 232.606,Z 1158.193,A -85,B 0,C 180,E1 6735.563,E2 6735.563} C_VEL
LIN {X 0,Y 233.973,Z 1153.484,A -85,B 0,C 180,E1 6730.529,E2 6730.529} C_VEL
LIN {X 0,Y 236.565,Z 1147.147,A -85,B 0,C 180,E1 6725.264,E2 6725.264} C_VEL
LIN {X 0,Y 240.53,Z 1138.988,A -85,B 0,C 180,E1 6720.077,E2 6720.077} C_VEL
LIN {X 0,Y 245.973,Z 1129.159,A -85,B 0,C 180,E1 6715.029,E2 6715.029} C_VEL
LIN {X 0,Y 252.197,Z 1118.5,A -85,B 0,C 180,E1 6710.629,E2 6710.629} C_VEL
LIN {X 0,Y 260.092,Z 1105.373,A -85,B 0,C 180,E1 6706.214,E2 6706.214} C_VEL
LIN {X 0,Y 268.455,Z 1091.401,A -85,B 0,C 180,E1 6702.386,E2 6702.386} C_VEL
LIN {X 0,Y 277.271,Z 1076.053,A -85,B 0,C 180,E1 6698.983,E2 6698.983} C_VEL
LIN {X 0,Y 286.5,Z 1059.308,A -85,B 0,C 180,E1 6695.937,E2 6695.937} C_VEL
LIN {X 0,Y 294.918,Z 1042.794,A -85,B 0,C 180,E1 6693.486,E2 6693.486} C_VEL
LIN {X 0,Y 304.292,Z 1022.764,A -85,B 0,C 180,E1 6691.056,E2 6691.056} C_VEL
LIN {X 0,Y 312.175,Z 1004.112,A -85,B 0,C 180,E1 6689.216,E2 6689.216} C_VEL
LIN {X 0,Y 319.675,Z 983.814,A -85,B 0,C 180,E1 6687.601,E2 6687.601} C_VEL
LIN {X 0,Y 326.224,Z 963.619,A -85,B 0,C 180,E1 6686.298,E2 6686.298} C_VEL
LIN {X 0,Y 331.866,Z 942.463,A -85,B 0,C 180,E1 6685.229,E2 6685.229} C_VEL
LIN {X 0,Y 336.806,Z 919.672,A -85,B 0,C 180,E1 6684.346,E2 6684.346} C_VEL
LIN {X 0,Y 340.276,Z 898.062,A -85,B 0,C 180,E1 6683.726,E2 6683.726} C_VEL
LIN {X 0,Y 343.451,Z 865.235,A -85,B 0,C 180,E1 6683.011,E2 6683.011} C_VEL
LIN {X 0,Y 357.564,Z 696.955,A -85,B 0,C 180,E1 6679.606,E2 6679.606} C_VEL
LIN {X 0,Y 352.175,Z 687.408,A -85,B 0,C 180,E1 6676.748,E2 6676.748} C_VEL
LIN {X 0,Y 347.331,Z 679.492,A -85,B 0,C 180,E1 6673.738,E2 6673.738} C_VEL
LIN {X 0,Y 343.74,Z 674.023,A -85,B 0,C 180,E1 6671.068,E2 6671.068} C_VEL
LIN {X 0,Y 341.612,Z 670.818,A -85,B 0,C 180,E1 6669.178,E2 6669.178} C_VEL
LIN {X 0,Y 338.723,Z 666.506,A -85,B 0,C 180,E1 6665.93,E2 6665.93} C_VEL
LIN {X 0,Y 335.787,Z 662.716,A -85,B 0,C 180,E1 6659.829,E2 6659.829} C_VEL
LIN {X 0,Y 335.503,Z 662.676,A -85,B 0,C 180,E1 6657.096,E2 6657.096} C_VEL
LIN {X 0,Y 337.273,Z 666.331,A -85,B 0,C 180,E1 6650.874,E2 6650.874} C_VEL
LIN {X 0,Y 339.99,Z 671.383,A -85,B 0,C 180,E1 6647.085,E2 6647.085} C_VEL
LIN {X 0,Y 342.855,Z 676.576,A -85,B 0,C 180,E1 6644.263,E2 6644.263} C_VEL
LIN {X 0,Y 346.541,Z 682.994,A -85,B 0,C 180,E1 6641.408,E2 6641.408} C_VEL
LIN {X 0,Y 351.968,Z 693.167,A -85,B 0,C 180,E1 6637.976,E2 6637.976} C_VEL
LIN {X 0,Y 355.793,Z 700.884,A -85,B 0,C 180,E1 6635.899,E2 6635.899} C_VEL
LIN {X 0,Y 340.283,Z 895.439,A -85,B 0,C 180,E1 6632.132,E2 6632.132} C_VEL
LIN {X 0,Y 337.006,Z 917.688,A -85,B 0,C 180,E1 6631.549,E2 6631.549} C_VEL
LIN {X 0,Y 332.559,Z 939.474,A -85,B 0,C 180,E1 6630.769,E2 6630.769} C_VEL
LIN {X 0,Y 327.349,Z 959.408,A -85,B 0,C 180,E1 6629.814,E2 6629.814} C_VEL
LIN {X 0,Y 320.672,Z 980.507,A -85,B 0,C 180,E1 6628.515,E2 6628.515} C_VEL
LIN {X 0,Y 313.491,Z 999.931,A -85,B 0,C 180,E1 6627.016,E2 6627.016} C_VEL
LIN {X 0,Y 305.549,Z 1018.408,A -85,B 0,C 180,E1 6625.221,E2 6625.221} C_VEL
LIN {X 0,Y 296.368,Z 1037.48,A -85,B 0,C 180,E1 6622.929,E2 6622.929} C_VEL
LIN {X 0,Y 287.409,Z 1054.393,A -85,B 0,C 180,E1 6620.405,E2 6620.405} C_VEL
LIN {X 0,Y 278.186,Z 1070.175,A -85,B 0,C 180,E1 6617.461,E2 6617.461} C_VEL
LIN {X 0,Y 269.003,Z 1084.981,A -85,B 0,C 180,E1 6614.032,E2 6614.032} C_VEL
LIN {X 0,Y 260.776,Z 1097.716,A -85,B 0,C 180,E1 6610.389,E2 6610.389} C_VEL
LIN {X 0,Y 253.194,Z 1109,A -85,B 0,C 180,E1 6606.324,E2 6606.324} C_VEL
LIN {X 0,Y 245.925,Z 1119.945,A -85,B 0,C 180,E1 6601.36,E2 6601.36} C_VEL
LIN {X 0,Y 240.529,Z 1128.488,A -85,B 0,C 180,E1 6596.41,E2 6596.41} C_VEL
LIN {X 0,Y 236.45,Z 1135.459,A -85,B 0,C 180,E1 6591.065,E2 6591.065} C_VEL
LIN {X 0,Y 233.875,Z 1140.716,A -85,B 0,C 180,E1 6585.625,E2 6585.625} C_VEL
LIN {X 0,Y 232.606,Z 1144.257,A -85,B 0,C 180,E1 6580.401,E2 6580.401} C_VEL
LIN {X 0,Y 232.118,Z 1146.208,A -85,B 0,C 180,E1 6575.438,E2 6575.438} C_VEL
LIN {X 0,Y 232.03,Z 1146.948,A -85,B 0,C 180,E1 6570.988,E2 6570.988} C_VEL
LIN {X 0,Y 232.07,Z 1146.62,A -85,B 0,C 180,E1 6566.047,E2 6566.047} C_VEL
LIN {X 0,Y 232.353,Z 1145.099,A -85,B 0,C 180,E1 6561.338,E2 6561.338} C_VEL
LIN {X 0,Y 233.318,Z 1142.175,A -85,B 0,C 180,E1 6556.114,E2 6556.114} C_VEL
LIN {X 0,Y 235.307,Z 1137.675,A -85,B 0,C 180,E1 6550.902,E2 6550.902} C_VEL
LIN {X 0,Y 239.061,Z 1130.879,A -85,B 0,C 180,E1 6545.175,E2 6545.175} C_VEL
LIN {X 0,Y 243.877,Z 1123.23,A -85,B 0,C 180,E1 6540.259,E2 6540.259} C_VEL
LIN {X 0,Y 250.257,Z 1113.47,A -85,B 0,C 180,E1 6535.435,E2 6535.435} C_VEL
LIN {X 0,Y 257.727,Z 1102.307,A -85,B 0,C 180,E1 6531.061,E2 6531.061} C_VEL
LIN {X 0,Y 266.019,Z 1089.806,A -85,B 0,C 180,E1 6527.132,E2 6527.132} C_VEL
LIN {X 0,Y 274.886,Z 1075.737,A -85,B 0,C 180,E1 6523.628,E2 6523.628} C_VEL
LIN {X 0,Y 284.309,Z 1059.909,A -85,B 0,C 180,E1 6520.455,E2 6520.455} C_VEL
LIN {X 0,Y 293.072,Z 1044.142,A -85,B 0,C 180,E1 6517.887,E2 6517.887} C_VEL
LIN {X 0,Y 301.841,Z 1026.578,A -85,B 0,C 180,E1 6515.587,E2 6515.587} C_VEL
LIN {X 0,Y 308.131,Z 1012.834,A -85,B 0,C 180,E1 6514.074,E2 6514.074} C_VEL
LIN {X 0,Y 299.438,Z 1018.391,A -85,B 0,C 180,E1 6512.748,E2 6512.748} C_VEL
LIN {X 0,Y 290.588,Z 1024.112,A -85,B 0,C 180,E1 6511.303,E2 6511.303} C_VEL
LIN {X 0,Y 289.751,Z 1024.579,A -85,B 0,C 180,E1 6511.148,E2 6511.148} C_VEL
LIN {X 0,Y 286.024,Z 1027.255,A -85,B 0,C 180,E1 6510.618,E2 6510.618} C_VEL
LIN {X 0,Y 276.224,Z 1035.896,A -85,B 0,C 180,E1 6509.73,E2 6509.73} C_VEL
LIN {X 0,Y 273.109,Z 1037.894,A -85,B 0,C 180,E1 6509.22,E2 6509.22} C_VEL
LIN {X 0,Y 272.641,Z 1038.109,A -85,B 0,C 180,E1 6509.108,E2 6509.108} C_VEL
LIN {X 0,Y 264.116,Z 1042.261,A -85,B 0,C 180,E1 6507.019,E2 6507.019} C_VEL
LIN {X 0,Y 254.624,Z 1046.419,A -85,B 0,C 180,E1 6504.104,E2 6504.104} C_VEL
LIN {X 0,Y 247.696,Z 1049.275,A -85,B 0,C 180,E1 6501.552,E2 6501.552} C_VEL
LIN {X 0,Y 244.838,Z 1050.396,A -85,B 0,C 180,E1 6500.312,E2 6500.312} C_VEL
LIN {X 0,Y 240.926,Z 1051.899,A -85,B 0,C 180,E1 6498.386,E2 6498.386} C_VEL
LIN {X 0,Y 236.231,Z 1053.809,A -85,B 0,C 180,E1 6495.717,E2 6495.717} C_VEL
LIN {X 0,Y 234.991,Z 1054.207,A -85,B 0,C 180,E1 6494.792,E2 6494.792} C_VEL
LIN {X 0,Y 232.065,Z 1055.541,A -85,B 0,C 180,E1 6492.694,E2 6492.694} C_VEL
LIN {X 0,Y 230.837,Z 1055.963,A -85,B 0,C 180,E1 6491.494,E2 6491.494} C_VEL
LIN {X 0,Y 228.535,Z 1057.101,A -85,B 0,C 180,E1 6489.317,E2 6489.317} C_VEL
LIN {X 0,Y 227.998,Z 1057.653,A -85,B 0,C 180,E1 6488.068,E2 6488.068} C_VEL
LIN {X 0,Y 227.857,Z 1063.991,A -85,B 0,C 180,E1 6484.027,E2 6484.027} C_VEL
LIN {X 0,Y 228.231,Z 1068.462,A -85,B 0,C 180,E1 6480.001,E2 6480.001} C_VEL
LIN {X 0,Y 229.208,Z 1071.371,A -85,B 0,C 180,E1 6475.748,E2 6475.748} C_VEL
LIN {X 0,Y 230.755,Z 1072.394,A -85,B 0,C 180,E1 6471.78,E2 6471.78} C_VEL
LIN {X 0,Y 232.984,Z 1071.682,A -85,B 0,C 180,E1 6467.862,E2 6467.862} C_VEL
LIN {X 0,Y 236.19,Z 1069.124,A -85,B 0,C 180,E1 6463.777,E2 6463.777} C_VEL
LIN {X 0,Y 240.011,Z 1064.926,A -85,B 0,C 180,E1 6460.026,E2 6460.026} C_VEL
LIN {X 0,Y 241.709,Z 1063.071,A -85,B 0,C 180,E1 6458.653,E2 6458.653} C_VEL
LIN {X 0,Y 249.708,Z 1061.692,A -85,B 0,C 180,E1 6455.392,E2 6455.392} C_VEL
LIN {X 0,Y 260.683,Z 1059.027,A -85,B 0,C 180,E1 6452.1,E2 6452.1} C_VEL
LIN {X 0,Y 274.091,Z 1054.708,A -85,B 0,C 180,E1 6449.046,E2 6449.046} C_VEL
LIN {X 0,Y 286.628,Z 1049.964,A -85,B 0,C 180,E1 6446.847,E2 6446.847} C_VEL
LIN {X 0,Y 276.928,Z 1067.48,A -85,B 0,C 180,E1 6443.975,E2 6443.975} C_VEL
LIN {X 0,Y 266.888,Z 1084.536,A -85,B 0,C 180,E1 6440.512,E2 6440.512} C_VEL
LIN {X 0,Y 257.81,Z 1099.316,A -85,B 0,C 180,E1 6436.813,E2 6436.813} C_VEL
LIN {X 0,Y 249.348,Z 1112.58,A -85,B 0,C 180,E1 6432.662,E2 6432.662} C_VEL
LIN {X 0,Y 241.246,Z 1125.442,A -85,B 0,C 180,E1 6427.665,E2 6427.665} C_VEL
LIN {X 0,Y 234.991,Z 1135.87,A -85,B 0,C 180,E1 6422.6,E2 6422.6} C_VEL
LIN {X 0,Y 230.109,Z 1144.657,A -85,B 0,C 180,E1 6417.145,E2 6417.145} C_VEL
LIN {X 0,Y 226.764,Z 1151.858,A -85,B 0,C 180,E1 6411.467,E2 6411.467} C_VEL
LIN {X 0,Y 224.976,Z 1156.816,A -85,B 0,C 180,E1 6406.26,E2 6406.26} C_VEL
LIN {X 0,Y 224.143,Z 1160.614,A -85,B 0,C 180,E1 6400.799,E2 6400.799} C_VEL
LIN {X 0,Y 223.98,Z 1162.648,A -85,B 0,C 180,E1 6395.893,E2 6395.893} C_VEL
LIN {X 0,Y 224.012,Z 1163.482,A -85,B 0,C 180,E1 6391.535,E2 6391.535} C_VEL
LIN {X 0,Y 223.99,Z 1163.356,A -85,B 0,C 180,E1 6387.186,E2 6387.186} C_VEL
LIN {X 0,Y 223.998,Z 1162.051,A -85,B 0,C 180,E1 6382.275,E2 6382.275} C_VEL
LIN {X 0,Y 224.365,Z 1159.293,A -85,B 0,C 180,E1 6377.125,E2 6377.125} C_VEL
LIN {X 0,Y 225.618,Z 1154.903,A -85,B 0,C 180,E1 6371.506,E2 6371.506} C_VEL
LIN {X 0,Y 228.078,Z 1148.759,A -85,B 0,C 180,E1 6365.94,E2 6365.94} C_VEL
LIN {X 0,Y 232.152,Z 1140.789,A -85,B 0,C 180,E1 6360.311,E2 6360.311} C_VEL
LIN {X 0,Y 237.313,Z 1131.823,A -85,B 0,C 180,E1 6355.334,E2 6355.334} C_VEL
LIN {X 0,Y 244.271,Z 1120.538,A -85,B 0,C 180,E1 6350.31,E2 6350.31} C_VEL
LIN {X 0,Y 252.322,Z 1107.912,A -85,B 0,C 180,E1 6345.779,E2 6345.779} C_VEL
LIN {X 0,Y 261.202,Z 1093.68,A -85,B 0,C 180,E1 6341.717,E2 6341.717} C_VEL
LIN {X 0,Y 271.217,Z 1077.162,A -85,B 0,C 180,E1 6337.915,E2 6337.915} C_VEL
LIN {X 0,Y 280.641,Z 1060.86,A -85,B 0,C 180,E1 6334.88,E2 6334.88} C_VEL
LIN {X 0,Y 289.777,Z 1043.614,A -85,B 0,C 180,E1 6332.289,E2 6332.289} C_VEL
LIN {X 0,Y 298.96,Z 1024.849,A -85,B 0,C 180,E1 6329.978,E2 6329.978} C_VEL
LIN {X 0,Y 306.707,Z 1007.2,A -85,B 0,C 180,E1 6328.209,E2 6328.209} C_VEL
LIN {X 0,Y 314.996,Z 985.919,A -85,B 0,C 180,E1 6326.475,E2 6326.475} C_VEL
LIN {X 0,Y 321.787,Z 965.74,A -85,B 0,C 180,E1 6325.161,E2 6325.161} C_VEL
LIN {X 0,Y 327.703,Z 944.609,A -85,B 0,C 180,E1 6324.077,E2 6324.077} C_VEL
LIN {X 0,Y 332.752,Z 922.684,A -85,B 0,C 180,E1 6323.205,E2 6323.205} C_VEL
LIN {X 0,Y 336.538,Z 900.189,A -85,B 0,C 180,E1 6322.553,E2 6322.553} C_VEL
LIN {X 0,Y 339.701,Z 869.886,A -85,B 0,C 180,E1 6321.884,E2 6321.884} C_VEL
LIN {X 0,Y 354.195,Z 701.749,A -85,B 0,C 180,E1 6318.495,E2 6318.495} C_VEL
LIN {X 0,Y 348.862,Z 692.339,A -85,B 0,C 180,E1 6315.458,E2 6315.458} C_VEL
LIN {X 0,Y 344.817,Z 685.632,A -85,B 0,C 180,E1 6312.731,E2 6312.731} C_VEL
LIN {X 0,Y 340.882,Z 679.24,A -85,B 0,C 180,E1 6309.454,E2 6309.454} C_VEL
LIN {X 0,Y 337.602,Z 674.377,A -85,B 0,C 180,E1 6305.779,E2 6305.779} C_VEL
LIN {X 0,Y 334.804,Z 670.668,A -85,B 0,C 180,E1 6299.828,E2 6299.828} C_VEL
LIN {X 0,Y 334.531,Z 670.631,A -85,B 0,C 180,E1 6297.087,E2 6297.087} C_VEL
LIN {X 0,Y 336.201,Z 674.273,A -85,B 0,C 180,E1 6291.017,E2 6291.017} C_VEL
LIN {X 0,Y 338.795,Z 679.249,A -85,B 0,C 180,E1 6287.298,E2 6287.298} C_VEL
LIN {X 0,Y 341.505,Z 684.301,A -85,B 0,C 180,E1 6284.548,E2 6284.548} C_VEL
LIN {X 0,Y 345.156,Z 690.928,A -85,B 0,C 180,E1 6281.637,E2 6281.637} C_VEL
LIN {X 0,Y 350.149,Z 700.621,A -85,B 0,C 180,E1 6278.385,E2 6278.385} C_VEL
LIN {X 0,Y 352.506,Z 705.745,A -85,B 0,C 180,E1 6277.019,E2 6277.019} C_VEL
LIN {X 0,Y 336.892,Z 895.383,A -85,B 0,C 180,E1 6273.362,E2 6273.362} C_VEL
LIN {X 0,Y 333.512,Z 917.766,A -85,B 0,C 180,E1 6272.783,E2 6272.783} C_VEL
LIN {X 0,Y 328.934,Z 939.609,A -85,B 0,C 180,E1 6272.011,E2 6272.011} C_VEL
LIN {X 0,Y 323.776,Z 958.888,A -85,B 0,C 180,E1 6271.103,E2 6271.103} C_VEL
LIN {X 0,Y 316.926,Z 980.109,A -85,B 0,C 180,E1 6269.818,E2 6269.818} C_VEL
LIN {X 0,Y 309.541,Z 999.604,A -85,B 0,C 180,E1 6268.336,E2 6268.336} C_VEL
LIN {X 0,Y 301.363,Z 1018.144,A -85,B 0,C 180,E1 6266.556,E2 6266.556} C_VEL
LIN {X 0,Y 292.207,Z 1036.689,A -85,B 0,C 180,E1 6264.358,E2 6264.358} C_VEL
LIN {X 0,Y 283.212,Z 1053.165,A -85,B 0,C 180,E1 6261.933,E2 6261.933} C_VEL
LIN {X 0,Y 273.866,Z 1068.723,A -85,B 0,C 180,E1 6259.09,E2 6259.09} C_VEL
LIN {X 0,Y 264.728,Z 1083.063,A -85,B 0,C 180,E1 6255.858,E2 6255.858} C_VEL
LIN {X 0,Y 255.957,Z 1096.004,A -85,B 0,C 180,E1 6252.214,E2 6252.214} C_VEL
LIN {X 0,Y 247.421,Z 1108.207,A -85,B 0,C 180,E1 6247.898,E2 6247.898} C_VEL
LIN {X 0,Y 240.238,Z 1118.486,A -85,B 0,C 180,E1 6243.324,E2 6243.324} C_VEL
LIN {X 0,Y 234.189,Z 1127.267,A -85,B 0,C 180,E1 6238.288,E2 6238.288} C_VEL
LIN {X 0,Y 229.515,Z 1134.603,A -85,B 0,C 180,E1 6232.813,E2 6232.813} C_VEL
LIN {X 0,Y 226.469,Z 1140.232,A -85,B 0,C 180,E1 6227.206,E2 6227.206} C_VEL
LIN {X 0,Y 224.845,Z 1143.95,A -85,B 0,C 180,E1 6221.804,E2 6221.804} C_VEL
LIN {X 0,Y 224.185,Z 1146.31,A -85,B 0,C 180,E1 6216.402,E2 6216.402} C_VEL
LIN {X 0,Y 224.036,Z 1147.196,A -85,B 0,C 180,E1 6211.534,E2 6211.534} C_VEL
LIN {X 0,Y 224.058,Z 1147.06,A -85,B 0,C 180,E1 6206.674,E2 6206.674} C_VEL
LIN {X 0,Y 224.337,Z 1145.605,A -85,B 0,C 180,E1 6201.542,E2 6201.542} C_VEL
LIN {X 0,Y 225.247,Z 1142.966,A -85,B 0,C 180,E1 6196.393,E2 6196.393} C_VEL
LIN {X 0,Y 227.354,Z 1138.455,A -85,B 0,C 180,E1 6190.741,E2 6190.741} C_VEL
LIN {X 0,Y 230.962,Z 1132.325,A -85,B 0,C 180,E1 6185.17,E2 6185.17} C_VEL
LIN {X 0,Y 235.948,Z 1124.714,A -85,B 0,C 180,E1 6179.997,E2 6179.997} C_VEL
LIN {X 0,Y 242.488,Z 1115.271,A -85,B 0,C 180,E1 6175.03,E2 6175.03} C_VEL
LIN {X 0,Y 250.151,Z 1104.474,A -85,B 0,C 180,E1 6170.541,E2 6170.541} C_VEL
LIN {X 0,Y 258.638,Z 1092.201,A -85,B 0,C 180,E1 6166.518,E2 6166.518} C_VEL
LIN {X 0,Y 267.718,Z 1078.554,A -85,B 0,C 180,E1 6162.944,E2 6162.944} C_VEL
LIN {X 0,Y 277.163,Z 1063.615,A -85,B 0,C 180,E1 6159.79,E2 6159.79} C_VEL
LIN {X 0,Y 286.413,Z 1047.617,A -85,B 0,C 180,E1 6157.09,E2 6157.09} C_VEL
LIN {X 0,Y 295.911,Z 1029.629,A -85,B 0,C 180,E1 6154.637,E2 6154.637} C_VEL
LIN {X 0,Y 298.763,Z 1023.723,A -85,B 0,C 180,E1 6153.904,E2 6153.904} C_VEL
LIN {X 0,Y 288.303,Z 1030.009,A -85,B 0,C 180,E1 6152.282,E2 6152.282} C_VEL
LIN {X 0,Y 274.878,Z 1037.122,A -85,B 0,C 180,E1 6149.65,E2 6149.65} C_VEL
LIN {X 0,Y 272.641,Z 1038.109,A -85,B 0,C 180,E1 6149.108,E2 6149.108} C_VEL
LIN {X 0,Y 267.629,Z 1040.807,A -85,B 0,C 180,E1 6148.006,E2 6148.006} C_VEL
LIN {X 0,Y 252.306,Z 1050.976,A -85,B 0,C 180,E1 6145.265,E2 6145.265} C_VEL
LIN {X 0,Y 248.87,Z 1052.821,A -85,B 0,C 180,E1 6144.373,E2 6144.373} C_VEL
LIN {X 0,Y 243.577,Z 1054.994,A -85,B 0,C 180,E1 6142.443,E2 6142.443} C_VEL
LIN {X 0,Y 236.494,Z 1057.613,A -85,B 0,C 180,E1 6139.256,E2 6139.256} C_VEL
LIN {X 0,Y 231.232,Z 1059.548,A -85,B 0,C 180,E1 6136.324,E2 6136.324} C_VEL
LIN {X 0,Y 229.101,Z 1060.35,A -85,B 0,C 180,E1 6134.922,E2 6134.922} C_VEL
LIN {X 0,Y 226.168,Z 1061.376,A -85,B 0,C 180,E1 6132.511,E2 6132.511} C_VEL
LIN {X 0,Y 223.196,Z 1062.771,A -85,B 0,C 180,E1 6129.802,E2 6129.802} C_VEL
LIN {X 0,Y 222.087,Z 1063.221,A -85,B 0,C 180,E1 6128.284,E2 6128.284} C_VEL
LIN {X 0,Y 220.161,Z 1064.329,A -85,B 0,C 180,E1 6125.473,E2 6125.473} C_VEL
LIN {X 0,Y 219.925,Z 1064.911,A -85,B 0,C 180,E1 6124.172,E2 6124.172} C_VEL
LIN {X 0,Y 220.365,Z 1069.882,A -85,B 0,C 180,E1 6119.741,E2 6119.741} C_VEL
LIN {X 0,Y 221.446,Z 1072.955,A -85,B 0,C 180,E1 6115.339,E2 6115.339} C_VEL
LIN {X 0,Y 223.153,Z 1074.144,A -85,B 0,C 180,E1 6111.238,E2 6111.238} C_VEL
LIN {X 0,Y 225.699,Z 1073.602,A -85,B 0,C 180,E1 6107.064,E2 6107.064} C_VEL
LIN {X 0,Y 229.33,Z 1071.124,A -85,B 0,C 180,E1 6102.755,E2 6102.755} C_VEL
LIN {X 0,Y 231.652,Z 1069.234,A -85,B 0,C 180,E1 6100.589,E2 6100.589} C_VEL
LIN {X 0,Y 239.213,Z 1068.47,A -85,B 0,C 180,E1 6096.866,E2 6096.866} C_VEL
LIN {X 0,Y 250.443,Z 1066.268,A -85,B 0,C 180,E1 6092.928,E2 6092.928} C_VEL
LIN {X 0,Y 263.945,Z 1062.666,A -85,B 0,C 180,E1 6089.496,E2 6089.496} C_VEL
LIN {X 0,Y 276.1,Z 1058.564,A -85,B 0,C 180,E1 6087.157,E2 6087.157} C_VEL
LIN {X 0,Y 277.297,Z 1058.223,A -85,B 0,C 180,E1 6086.918,E2 6086.918} C_VEL
LIN {X 0,Y 267.345,Z 1075.014,A -85,B 0,C 180,E1 6083.885,E2 6083.885} C_VEL
LIN {X 0,Y 257.802,Z 1090.281,A -85,B 0,C 180,E1 6080.503,E2 6080.503} C_VEL
LIN {X 0,Y 248.708,Z 1104.048,A -85,B 0,C 180,E1 6076.691,E2 6076.691} C_VEL
LIN {X 0,Y 239.665,Z 1117.587,A -85,B 0,C 180,E1 6072.048,E2 6072.048} C_VEL
LIN {X 0,Y 232.088,Z 1129.096,A -85,B 0,C 180,E1 6067.095,E2 6067.095} C_VEL
LIN {X 0,Y 225.924,Z 1138.824,A -85,B 0,C 180,E1 6061.78,E2 6061.78} C_VEL
LIN {X 0,Y 221.206,Z 1147.207,A -85,B 0,C 180,E1 6056.005,E2 6056.005} C_VEL
LIN {X 0,Y 218.357,Z 1153.167,A -85,B 0,C 180,E1 6050.646,E2 6050.646} C_VEL
LIN {X 0,Y 216.638,Z 1158.158,A -85,B 0,C 180,E1 6044.705,E2 6044.705} C_VEL
LIN {X 0,Y 216.078,Z 1161.053,A -85,B 0,C 180,E1 6039.589,E2 6039.589} C_VEL
LIN {X 0,Y 215.992,Z 1162.722,A -85,B 0,C 180,E1 6034.78,E2 6034.78} C_VEL
LIN {X 0,Y 216.014,Z 1163.309,A -85,B 0,C 180,E1 6029.735,E2 6029.735} C_VEL
LIN {X 0,Y 215.989,Z 1162.642,A -85,B 0,C 180,E1 6024.954,E2 6024.954} C_VEL
LIN {X 0,Y 216.086,Z 1160.919,A -85,B 0,C 180,E1 6020.142,E2 6020.142} C_VEL
LIN {X 0,Y 216.798,Z 1157.591,A -85,B 0,C 180,E1 6014.485,E2 6014.485} C_VEL
LIN {X 0,Y 218.518,Z 1152.764,A -85,B 0,C 180,E1 6008.973,E2 6008.973} C_VEL
LIN {X 0,Y 221.746,Z 1146.163,A -85,B 0,C 180,E1 6003.198,E2 6003.198} C_VEL
LIN {X 0,Y 226.435,Z 1137.935,A -85,B 0,C 180,E1 5997.704,E2 5997.704} C_VEL
LIN {X 0,Y 233.205,Z 1127.261,A -85,B 0,C 180,E1 5992.081,E2 5992.081} C_VEL
LIN {X 0,Y 241.103,Z 1115.458,A -85,B 0,C 180,E1 5987.147,E2 5987.147} C_VEL
LIN {X 0,Y 249.657,Z 1102.521,A -85,B 0,C 180,E1 5982.87,E2 5982.87} C_VEL
LIN {X 0,Y 259.43,Z 1087.55,A -85,B 0,C 180,E1 5978.874,E2 5978.874} C_VEL
LIN {X 0,Y 268.807,Z 1072.522,A -85,B 0,C 180,E1 5975.636,E2 5975.636} C_VEL
LIN {X 0,Y 278.636,Z 1055.627,A -85,B 0,C 180,E1 5972.69,E2 5972.69} C_VEL
LIN {X 0,Y 288.09,Z 1038.203,A -85,B 0,C 180,E1 5970.209,E2 5970.209} C_VEL
LIN {X 0,Y 297.342,Z 1019.14,A -85,B 0,C 180,E1 5968.03,E2 5968.03} C_VEL
LIN {X 0,Y 306.268,Z 998.574,A -85,B 0,C 180,E1 5966.132,E2 5966.132} C_VEL
LIN {X 0,Y 314.022,Z 978.18,A -85,B 0,C 180,E1 5964.626,E2 5964.626} C_VEL
LIN {X 0,Y 320.815,Z 956.89,A -85,B 0,C 180,E1 5963.386,E2 5963.386} C_VEL
LIN {X 0,Y 326.758,Z 934.465,A -85,B 0,C 180,E1 5962.366,E2 5962.366} C_VEL
LIN {X 0,Y 331.256,Z 912.681,A -85,B 0,C 180,E1 5961.632,E2 5961.632} C_VEL
LIN {X 0,Y 334.694,Z 888.845,A -85,B 0,C 180,E1 5961.033,E2 5961.033} C_VEL
LIN {X 0,Y 350.975,Z 706.787,A -85,B 0,C 180,E1 5957.383,E2 5957.383} C_VEL
LIN {X 0,Y 346.093,Z 697.899,A -85,B 0,C 180,E1 5954.385,E2 5954.385} C_VEL
LIN {X 0,Y 341.715,Z 690.552,A -85,B 0,C 180,E1 5951.134,E2 5951.134} C_VEL
LIN {X 0,Y 338.925,Z 686.183,A -85,B 0,C 180,E1 5948.567,E2 5948.567} C_VEL
LIN {X 0,Y 336.366,Z 682.12,A -85,B 0,C 180,E1 5945.458,E2 5945.458} C_VEL
LIN {X 0,Y 333.795,Z 678.561,A -85,B 0,C 180,E1 5939.656,E2 5939.656} C_VEL
LIN {X 0,Y 333.555,Z 678.587,A -85,B 0,C 180,E1 5937.079,E2 5937.079} C_VEL
LIN {X 0,Y 335.132,Z 682.214,A -85,B 0,C 180,E1 5931.161,E2 5931.161} C_VEL
LIN {X 0,Y 337.538,Z 686.96,A -85,B 0,C 180,E1 5927.598,E2 5927.598} C_VEL
LIN {X 0,Y 340.255,Z 692.191,A -85,B 0,C 180,E1 5924.751,E2 5924.751} C_VEL
LIN {X 0,Y 344.276,Z 699.843,A -85,B 0,C 180,E1 5921.501,E2 5921.501} C_VEL
LIN {X 0,Y 349.004,Z 709.413,A -85,B 0,C 180,E1 5918.399,E2 5918.399} C_VEL
LIN {X 0,Y 349.377,Z 710.433,A -85,B 0,C 180,E1 5918.163,E2 5918.163} C_VEL
LIN {X 0,Y 333.666,Z 895.266,A -85,B 0,C 180,E1 5914.619,E2 5914.619} C_VEL
LIN {X 0,Y 330.219,Z 917.611,A -85,B 0,C 180,E1 5914.048,E2 5914.048} C_VEL
LIN {X 0,Y 325.467,Z 939.743,A -85,B 0,C 180,E1 5913.279,E2 5913.279} C_VEL
LIN {X 0,Y 320.001,Z 959.639,A -85,B 0,C 180,E1 5912.352,E2 5912.352} C_VEL
LIN {X 0,Y 312.983,Z 980.703,A -85,B 0,C 180,E1 5911.084,E2 5911.084} C_VEL
LIN {X 0,Y 305.407,Z 1000.122,A -85,B 0,C 180,E1 5909.617,E2 5909.617} C_VEL
LIN {X 0,Y 297.132,Z 1018.334,A -85,B 0,C 180,E1 5907.881,E2 5907.881} C_VEL
LIN {X 0,Y 287.573,Z 1037.094,A -85,B 0,C 180,E1 5905.666,E2 5905.666} C_VEL
LIN {X 0,Y 278.29,Z 1053.552,A -85,B 0,C 180,E1 5903.246,E2 5903.246} C_VEL
LIN {X 0,Y 268.613,Z 1069.077,A -85,B 0,C 180,E1 5900.401,E2 5900.401} C_VEL
LIN {X 0,Y 259.112,Z 1083.397,A -85,B 0,C 180,E1 5897.153,E2 5897.153} C_VEL
LIN {X 0,Y 249.962,Z 1096.333,A -85,B 0,C 180,E1 5893.473,E2 5893.473} C_VEL
LIN {X 0,Y 241.009,Z 1108.521,A -85,B 0,C 180,E1 5889.094,E2 5889.094} C_VEL
LIN {X 0,Y 233.433,Z 1118.793,A -85,B 0,C 180,E1 5884.43,E2 5884.43} C_VEL
LIN {X 0,Y 227.009,Z 1127.574,A -85,B 0,C 180,E1 5879.268,E2 5879.268} C_VEL
LIN {X 0,Y 222.005,Z 1134.903,A -85,B 0,C 180,E1 5873.63,E2 5873.63} C_VEL
LIN {X 0,Y 218.71,Z 1140.528,A -85,B 0,C 180,E1 5867.836,E2 5867.836} C_VEL
LIN {X 0,Y 216.94,Z 1144.245,A -85,B 0,C 180,E1 5862.24,E2 5862.24} C_VEL
LIN {X 0,Y 216.21,Z 1146.602,A -85,B 0,C 180,E1 5856.639,E2 5856.639} C_VEL
LIN {X 0,Y 216.041,Z 1147.465,A -85,B 0,C 180,E1 5851.856,E2 5851.856} C_VEL
LIN {X 0,Y 216.05,Z 1147.412,A -85,B 0,C 180,E1 5847.347,E2 5847.347} C_VEL
LIN {X 0,Y 216.303,Z 1146.218,A -85,B 0,C 180,E1 5842.029,E2 5842.029} C_VEL
LIN {X 0,Y 217.172,Z 1143.711,A -85,B 0,C 180,E1 5836.691,E2 5836.691} C_VEL
LIN {X 0,Y 219.404,Z 1139.236,A -85,B 0,C 180,E1 5830.569,E2 5830.569} C_VEL
LIN {X 0,Y 223.142,Z 1133.292,A -85,B 0,C 180,E1 5824.806,E2 5824.806} C_VEL
LIN {X 0,Y 228.307,Z 1125.795,A -85,B 0,C 180,E1 5819.468,E2 5819.468} C_VEL
LIN {X 0,Y 235.45,Z 1116.078,A -85,B 0,C 180,E1 5814.124,E2 5814.124} C_VEL
LIN {X 0,Y 243.451,Z 1105.405,A -85,B 0,C 180,E1 5809.54,E2 5809.54} C_VEL
LIN {X 0,Y 252.27,Z 1093.205,A -85,B 0,C 180,E1 5805.45,E2 5805.45} C_VEL
LIN {X 0,Y 262.234,Z 1078.893,A -85,B 0,C 180,E1 5801.641,E2 5801.641} C_VEL
LIN {X 0,Y 272.033,Z 1063.978,A -85,B 0,C 180,E1 5798.474,E2 5798.474} C_VEL
LIN {X 0,Y 281.6,Z 1047.995,A -85,B 0,C 180,E1 5795.774,E2 5795.774} C_VEL
LIN {X 0,Y 289.265,Z 1034.149,A -85,B 0,C 180,E1 5793.815,E2 5793.815} C_VEL
LIN {X 0,Y 272.244,Z 1042.783,A -85,B 0,C 180,E1 5790.698,E2 5790.698} C_VEL
LIN {X 0,Y 260.498,Z 1048.084,A -85,B 0,C 180,E1 5787.922,E2 5787.922} C_VEL
LIN {X 0,Y 250.687,Z 1052.128,A -85,B 0,C 180,E1 5785.011,E2 5785.011} C_VEL
LIN {X 0,Y 248.87,Z 1052.821,A -85,B 0,C 180,E1 5784.373,E2 5784.373} C_VEL
LIN {X 0,Y 242.714,Z 1056.283,A -85,B 0,C 180,E1 5782.705,E2 5782.705} C_VEL
LIN {X 0,Y 232.336,Z 1062.479,A -85,B 0,C 180,E1 5779.938,E2 5779.938} C_VEL
LIN {X 0,Y 228.2,Z 1064.504,A -85,B 0,C 180,E1 5778.242,E2 5778.242} C_VEL
LIN {X 0,Y 227.976,Z 1064.586,A -85,B 0,C 180,E1 5778.118,E2 5778.118} C_VEL
LIN {X 0,Y 223.943,Z 1065.989,A -85,B 0,C 180,E1 5775.539,E2 5775.539} C_VEL
LIN {X 0,Y 219.584,Z 1067.581,A -85,B 0,C 180,E1 5772.091,E2 5772.091} C_VEL
LIN {X 0,Y 217.067,Z 1068.489,A -85,B 0,C 180,E1 5769.278,E2 5769.278} C_VEL
LIN {X 0,Y 214.509,Z 1069.815,A -85,B 0,C 180,E1 5765.886,E2 5765.886} C_VEL
LIN {X 0,Y 213.518,Z 1070.449,A -85,B 0,C 180,E1 5763.76,E2 5763.76} C_VEL
LIN {X 0,Y 212.72,Z 1072.236,A -85,B 0,C 180,E1 5758.385,E2 5758.385} C_VEL
LIN {X 0,Y 214.095,Z 1075.052,A -85,B 0,C 180,E1 5753.835,E2 5753.835} C_VEL
LIN {X 0,Y 216.32,Z 1075.992,A -85,B 0,C 180,E1 5749.346,E2 5749.346} C_VEL
LIN {X 0,Y 219.487,Z 1075.102,A -85,B 0,C 180,E1 5744.951,E2 5744.951} C_VEL
LIN {X 0,Y 221.957,Z 1074.944,A -85,B 0,C 180,E1 5742.705,E2 5742.705} C_VEL
LIN {X 0,Y 230.444,Z 1074.382,A -85,B 0,C 180,E1 5737.823,E2 5737.823} C_VEL
LIN {X 0,Y 240.409,Z 1072.966,A -85,B 0,C 180,E1 5733.843,E2 5733.843} C_VEL
LIN {X 0,Y 253.216,Z 1070.209,A -85,B 0,C 180,E1 5730.164,E2 5730.164} C_VEL
LIN {X 0,Y 267.24,Z 1066.133,A -85,B 0,C 180,E1 5727.146,E2 5727.146} C_VEL
LIN {X 0,Y 267.869,Z 1066.045,A -85,B 0,C 180,E1 5726.989,E2 5726.989} C_VEL
LIN {X 0,Y 257.724,Z 1082.097,A -85,B 0,C 180,E1 5723.799,E2 5723.799} C_VEL
LIN {X 0,Y 248.206,Z 1096.254,A -85,B 0,C 180,E1 5720.302,E2 5720.302} C_VEL
LIN {X 0,Y 238.186,Z 1110.609,A -85,B 0,C 180,E1 5715.876,E2 5715.876} C_VEL
LIN {X 0,Y 229.533,Z 1122.949,A -85,B 0,C 180,E1 5711.098,E2 5711.098} C_VEL
LIN {X 0,Y 222.089,Z 1133.625,A -85,B 0,C 180,E1 5705.822,E2 5705.822} C_VEL
LIN {X 0,Y 216.061,Z 1142.929,A -85,B 0,C 180,E1 5699.986,E2 5699.986} C_VEL
LIN {X 0,Y 212.173,Z 1149.77,A -85,B 0,C 180,E1 5694.5,E2 5694.5} C_VEL
LIN {X 0,Y 209.478,Z 1155.663,A -85,B 0,C 180,E1 5688.226,E2 5688.226} C_VEL
LIN {X 0,Y 208.342,Z 1159.395,A -85,B 0,C 180,E1 5682.754,E2 5682.754} C_VEL
LIN {X 0,Y 207.99,Z 1161.842,A -85,B 0,C 180,E1 5677.18,E2 5677.18} C_VEL
LIN {X 0,Y 208.008,Z 1162.827,A -85,B 0,C 180,E1 5672.48,E2 5672.48} C_VEL
LIN {X 0,Y 208.019,Z 1162.874,A -85,B 0,C 180,E1 5668.072,E2 5668.072} C_VEL
LIN {X 0,Y 208,Z 1161.983,A -85,B 0,C 180,E1 5663.375,E2 5663.375} C_VEL
LIN {X 0,Y 208.278,Z 1159.718,A -85,B 0,C 180,E1 5657.806,E2 5657.806} C_VEL
LIN {X 0,Y 209.35,Z 1155.976,A -85,B 0,C 180,E1 5652.202,E2 5652.202} C_VEL
LIN {X 0,Y 211.873,Z 1150.376,A -85,B 0,C 180,E1 5646.056,E2 5646.056} C_VEL
LIN {X 0,Y 215.831,Z 1143.26,A -85,B 0,C 180,E1 5640.285,E2 5640.285} C_VEL
LIN {X 0,Y 221.772,Z 1134.053,A -85,B 0,C 180,E1 5634.437,E2 5634.437} C_VEL
LIN {X 0,Y 228.779,Z 1123.912,A -85,B 0,C 180,E1 5629.368,E2 5629.368} C_VEL
LIN {X 0,Y 237.245,Z 1111.845,A -85,B 0,C 180,E1 5624.582,E2 5624.582} C_VEL
LIN {X 0,Y 246.618,Z 1098.534,A -85,B 0,C 180,E1 5620.341,E2 5620.341} C_VEL
LIN {X 0,Y 256.547,Z 1083.721,A -85,B 0,C 180,E1 5616.596,E2 5616.596} C_VEL
LIN {X 0,Y 267.44,Z 1066.587,A -85,B 0,C 180,E1 5613.127,E2 5613.127} C_VEL
LIN {X 0,Y 277.541,Z 1049.589,A -85,B 0,C 180,E1 5610.366,E2 5610.366} C_VEL
LIN {X 0,Y 287.07,Z 1031.783,A -85,B 0,C 180,E1 5608.047,E2 5608.047} C_VEL
LIN {X 0,Y 296.441,Z 1012.532,A -85,B 0,C 180,E1 5606.006,E2 5606.006} C_VEL
LIN {X 0,Y 304.242,Z 994.37,A -85,B 0,C 180,E1 5604.449,E2 5604.449} C_VEL
LIN {X 0,Y 312.236,Z 973.064,A -85,B 0,C 180,E1 5602.979,E2 5602.979} C_VEL
LIN {X 0,Y 318.449,Z 953.534,A -85,B 0,C 180,E1 5601.905,E2 5601.905} C_VEL
LIN {X 0,Y 324.31,Z 930.938,A -85,B 0,C 180,E1 5600.94,E2 5600.94} C_VEL
LIN {X 0,Y 328.93,Z 908.195,A -85,B 0,C 180,E1 5600.222,E2 5600.222} C_VEL
LIN {X 0,Y 331.993,Z 885.399,A -85,B 0,C 180,E1 5599.685,E2 5599.685} C_VEL
LIN {X 0,Y 347.848,Z 711.777,A -85,B 0,C 180,E1 5596.228,E2 5596.228} C_VEL
LIN {X 0,Y 343.257,Z 703.376,A -85,B 0,C 180,E1 5593.175,E2 5593.175} C_VEL
LIN {X 0,Y 339.638,Z 697.212,A -85,B 0,C 180,E1 5590.259,E2 5590.259} C_VEL
LIN {X 0,Y 337.517,Z 693.756,A -85,B 0,C 180,E1 5588.174,E2 5588.174} C_VEL
LIN {X 0,Y 335.259,Z 689.992,A -85,B 0,C 180,E1 5585.304,E2 5585.304} C_VEL
LIN {X 0,Y 332.789,Z 686.456,A -85,B 0,C 180,E1 5579.483,E2 5579.483} C_VEL
LIN {X 0,Y 332.58,Z 686.608,A -85,B 0,C 180,E1 5576.897,E2 5576.897} C_VEL
LIN {X 0,Y 334.067,Z 690.152,A -85,B 0,C 180,E1 5571.306,E2 5571.306} C_VEL
LIN {X 0,Y 336.288,Z 694.669,A -85,B 0,C 180,E1 5567.9,E2 5567.9} C_VEL
LIN {X 0,Y 339.099,Z 700.234,A -85,B 0,C 180,E1 5564.873,E2 5564.873} C_VEL
LIN {X 0,Y 342.779,Z 707.56,A -85,B 0,C 180,E1 5561.813,E2 5561.813} C_VEL
LIN {X 0,Y 346.369,Z 715.23,A -85,B 0,C 180,E1 5559.325,E2 5559.325} C_VEL
LIN {X 0,Y 330.589,Z 895.275,A -85,B 0,C 180,E1 5555.896,E2 5555.896} C_VEL
LIN {X 0,Y 327.052,Z 917.65,A -85,B 0,C 180,E1 5555.333,E2 5555.333} C_VEL
LIN {X 0,Y 322.163,Z 939.874,A -85,B 0,C 180,E1 5554.575,E2 5554.575} C_VEL
LIN {X 0,Y 316.382,Z 960.389,A -85,B 0,C 180,E1 5553.63,E2 5553.63} C_VEL
LIN {X 0,Y 309.196,Z 981.295,A -85,B 0,C 180,E1 5552.381,E2 5552.381} C_VEL
LIN {X 0,Y 301.428,Z 1000.619,A -85,B 0,C 180,E1 5550.933,E2 5550.933} C_VEL
LIN {X 0,Y 292.815,Z 1019.03,A -85,B 0,C 180,E1 5549.189,E2 5549.189} C_VEL
LIN {X 0,Y 282.756,Z 1038.097,A -85,B 0,C 180,E1 5546.936,E2 5546.936} C_VEL
LIN {X 0,Y 272.877,Z 1055.001,A -85,B 0,C 180,E1 5544.434,E2 5544.434} C_VEL
LIN {X 0,Y 262.903,Z 1070.339,A -85,B 0,C 180,E1 5541.578,E2 5541.578} C_VEL
LIN {X 0,Y 252.524,Z 1085.233,A -85,B 0,C 180,E1 5538.106,E2 5538.106} C_VEL
LIN {X 0,Y 242.797,Z 1098.441,A -85,B 0,C 180,E1 5534.229,E2 5534.229} C_VEL
LIN {X 0,Y 233.846,Z 1109.95,A -85,B 0,C 180,E1 5529.893,E2 5529.893} C_VEL
LIN {X 0,Y 225.639,Z 1120.426,A -85,B 0,C 180,E1 5524.864,E2 5524.864} C_VEL
LIN {X 0,Y 219.067,Z 1129.045,A -85,B 0,C 180,E1 5519.533,E2 5519.533} C_VEL
LIN {X 0,Y 213.953,Z 1136.074,A -85,B 0,C 180,E1 5513.697,E2 5513.697} C_VEL
LIN {X 0,Y 210.505,Z 1141.606,A -85,B 0,C 180,E1 5507.412,E2 5507.412} C_VEL
LIN {X 0,Y 208.767,Z 1145.287,A -85,B 0,C 180,E1 5501.324,E2 5501.324} C_VEL
LIN {X 0,Y 208.155,Z 1147.146,A -85,B 0,C 180,E1 5495.789,E2 5495.789} C_VEL
LIN {X 0,Y 208.046,Z 1147.841,A -85,B 0,C 180,E1 5490.826,E2 5490.826} C_VEL
LIN {X 0,Y 208.11,Z 1147.43,A -85,B 0,C 180,E1 5485.315,E2 5485.315} C_VEL
LIN {X 0,Y 208.545,Z 1145.87,A -85,B 0,C 180,E1 5480.061,E2 5480.061} C_VEL
LIN {X 0,Y 209.954,Z 1142.671,A -85,B 0,C 180,E1 5473.966,E2 5473.966} C_VEL
LIN {X 0,Y 212.668,Z 1138.081,A -85,B 0,C 180,E1 5468.197,E2 5468.197} C_VEL
LIN {X 0,Y 217.171,Z 1131.572,A -85,B 0,C 180,E1 5462.289,E2 5462.289} C_VEL
LIN {X 0,Y 223.183,Z 1123.71,A -85,B 0,C 180,E1 5456.868,E2 5456.868} C_VEL
LIN {X 0,Y 230.829,Z 1113.895,A -85,B 0,C 180,E1 5451.726,E2 5451.726} C_VEL
LIN {X 0,Y 239.583,Z 1102.642,A -85,B 0,C 180,E1 5447.136,E2 5447.136} C_VEL
LIN {X 0,Y 249.149,Z 1090.05,A -85,B 0,C 180,E1 5443.081,E2 5443.081} C_VEL
LIN {X 0,Y 258.626,Z 1076.751,A -85,B 0,C 180,E1 5439.705,E2 5439.705} C_VEL
LIN {X 0,Y 269.413,Z 1060.565,A -85,B 0,C 180,E1 5436.428,E2 5436.428} C_VEL
LIN {X 0,Y 279.596,Z 1043.953,A -85,B 0,C 180,E1 5433.753,E2 5433.753} C_VEL
LIN {X 0,Y 279.805,Z 1043.365,A -85,B 0,C 180,E1 5433.632,E2 5433.632} C_VEL
LIN {X 0,Y 269.563,Z 1048.303,A -85,B 0,C 180,E1 5431.784,E2 5431.784} C_VEL
LIN {X 0,Y 256.99,Z 1053.732,A -85,B 0,C 180,E1 5428.907,E2 5428.907} C_VEL
LIN {X 0,Y 246.727,Z 1057.744,A -85,B 0,C 180,E1 5425.956,E2 5425.956} C_VEL
LIN {X 0,Y 238.828,Z 1060.663,A -85,B 0,C 180,E1 5423.175,E2 5423.175} C_VEL
LIN {X 0,Y 231.551,Z 1063.234,A -85,B 0,C 180,E1 5419.946,E2 5419.946} C_VEL
LIN {X 0,Y 227.976,Z 1064.586,A -85,B 0,C 180,E1 5418.118,E2 5418.118} C_VEL
LIN {X 0,Y 224.979,Z 1066.221,A -85,B 0,C 180,E1 5416.872,E2 5416.872} C_VEL
LIN {X 0,Y 216.579,Z 1071.673,A -85,B 0,C 180,E1 5414.191,E2 5414.191} C_VEL
LIN {X 0,Y 214.951,Z 1072.56,A -85,B 0,C 180,E1 5413.324,E2 5413.324} C_VEL
LIN {X 0,Y 211.774,Z 1073.809,A -85,B 0,C 180,E1 5410.336,E2 5410.336} C_VEL
LIN {X 0,Y 208.564,Z 1075.297,A -85,B 0,C 180,E1 5405.779,E2 5405.779} C_VEL
LIN {X 0,Y 206.642,Z 1077.026,A -85,B 0,C 180,E1 5399.724,E2 5399.724} C_VEL
LIN {X 0,Y 208.465,Z 1079.381,A -85,B 0,C 180,E1 5390.337,E2 5390.337} C_VEL
LIN {X 0,Y 214.085,Z 1080.108,A -85,B 0,C 180,E1 5384.006,E2 5384.006} C_VEL
LIN {X 0,Y 219.692,Z 1080.167,A -85,B 0,C 180,E1 5380.042,E2 5380.042} C_VEL
LIN {X 0,Y 228.945,Z 1079.438,A -85,B 0,C 180,E1 5375.489,E2 5375.489} C_VEL
LIN {X 0,Y 241.25,Z 1077.344,A -85,B 0,C 180,E1 5371.266,E2 5371.266} C_VEL
LIN {X 0,Y 255.229,Z 1074.061,A -85,B 0,C 180,E1 5367.807,E2 5367.807} C_VEL
LIN {X 0,Y 258.481,Z 1073.342,A -85,B 0,C 180,E1 5367.077,E2 5367.077} C_VEL
LIN {X 0,Y 247.889,Z 1088.995,A -85,B 0,C 180,E1 5363.636,E2 5363.636} C_VEL
LIN {X 0,Y 237.505,Z 1103.379,A -85,B 0,C 180,E1 5359.64,E2 5359.64} C_VEL
LIN {X 0,Y 227.683,Z 1116.669,A -85,B 0,C 180,E1 5354.994,E2 5354.994} C_VEL
LIN {X 0,Y 219.302,Z 1127.922,A -85,B 0,C 180,E1 5350.006,E2 5350.006} C_VEL
LIN {X 0,Y 212.166,Z 1137.778,A -85,B 0,C 180,E1 5344.438,E2 5344.438} C_VEL
LIN {X 0,Y 206.788,Z 1145.947,A -85,B 0,C 180,E1 5338.6,E2 5338.6} C_VEL
LIN {X 0,Y 202.974,Z 1152.562,A -85,B 0,C 180,E1 5332.291,E2 5332.291} C_VEL
LIN {X 0,Y 200.85,Z 1157.563,A -85,B 0,C 180,E1 5325.891,E2 5325.891} C_VEL
LIN {X 0,Y 200.109,Z 1160.464,A -85,B 0,C 180,E1 5320.363,E2 5320.363} C_VEL
LIN {X 0,Y 199.991,Z 1162.065,A -85,B 0,C 180,E1 5315.451,E2 5315.451} C_VEL
LIN {X 0,Y 200.033,Z 1162.745,A -85,B 0,C 180,E1 5310,E2 5310} C_VEL
LIN {X 0,Y 199.995,Z 1162.131,A -85,B 0,C 180,E1 5304.837,E2 5304.837} C_VEL
LIN {X 0,Y 200.099,Z 1160.541,A -85,B 0,C 180,E1 5299.853,E2 5299.853} C_VEL
LIN {X 0,Y 200.789,Z 1157.717,A -85,B 0,C 180,E1 5294.401,E2 5294.401} C_VEL
LIN {X 0,Y 202.889,Z 1152.704,A -85,B 0,C 180,E1 5287.89,E2 5287.89} C_VEL
LIN {X 0,Y 206.571,Z 1146.243,A -85,B 0,C 180,E1 5281.683,E2 5281.683} C_VEL
LIN {X 0,Y 211.865,Z 1138.153,A -85,B 0,C 180,E1 5275.833,E2 5275.833} C_VEL
LIN {X 0,Y 218.919,Z 1128.399,A -85,B 0,C 180,E1 5270.252,E2 5270.252} C_VEL
LIN {X 0,Y 227.22,Z 1117.193,A -85,B 0,C 180,E1 5265.246,E2 5265.246} C_VEL
LIN {X 0,Y 237.226,Z 1103.655,A -85,B 0,C 180,E1 5260.471,E2 5260.471} C_VEL
LIN {X 0,Y 247.501,Z 1089.438,A -85,B 0,C 180,E1 5256.493,E2 5256.493} C_VEL
LIN {X 0,Y 258.151,Z 1073.687,A -85,B 0,C 180,E1 5253.014,E2 5253.014} C_VEL
LIN {X 0,Y 269.307,Z 1056.001,A -85,B 0,C 180,E1 5249.897,E2 5249.897} C_VEL
LIN {X 0,Y 279.813,Z 1037.888,A -85,B 0,C 180,E1 5247.346,E2 5247.346} C_VEL
LIN {X 0,Y 289.578,Z 1018.943,A -85,B 0,C 180,E1 5245.225,E2 5245.225} C_VEL
LIN {X 0,Y 299.149,Z 998.048,A -85,B 0,C 180,E1 5243.352,E2 5243.352} C_VEL
LIN {X 0,Y 307.56,Z 976.951,A -85,B 0,C 180,E1 5241.852,E2 5241.852} C_VEL
LIN {X 0,Y 314.52,Z 955.914,A -85,B 0,C 180,E1 5240.683,E2 5240.683} C_VEL
LIN {X 0,Y 320.868,Z 932.579,A -85,B 0,C 180,E1 5239.679,E2 5239.679} C_VEL
LIN {X 0,Y 325.637,Z 910.053,A -85,B 0,C 180,E1 5238.967,E2 5238.967} C_VEL
LIN {X 0,Y 328.922,Z 886.881,A -85,B 0,C 180,E1 5238.42,E2 5238.42} C_VEL
LIN {X 0,Y 344.871,Z 716.927,A -85,B 0,C 180,E1 5235.067,E2 5235.067} C_VEL
LIN {X 0,Y 340.88,Z 709.428,A -85,B 0,C 180,E1 5232.191,E2 5232.191} C_VEL
LIN {X 0,Y 337.648,Z 703.844,A -85,B 0,C 180,E1 5229.373,E2 5229.373} C_VEL
LIN {X 0,Y 335.84,Z 700.882,A -85,B 0,C 180,E1 5227.441,E2 5227.441} C_VEL
LIN {X 0,Y 334.039,Z 697.734,A -85,B 0,C 180,E1 5224.979,E2 5224.979} C_VEL
LIN {X 0,Y 331.813,Z 694.407,A -85,B 0,C 180,E1 5219.482,E2 5219.482} C_VEL
LIN {X 0,Y 331.603,Z 694.571,A -85,B 0,C 180,E1 5216.888,E2 5216.888} C_VEL
LIN {X 0,Y 332.966,Z 697.971,A -85,B 0,C 180,E1 5211.538,E2 5211.538} C_VEL
LIN {X 0,Y 335.056,Z 702.413,A -85,B 0,C 180,E1 5208.183,E2 5208.183} C_VEL
LIN {X 0,Y 337.946,Z 708.266,A -85,B 0,C 180,E1 5204.996,E2 5204.996} C_VEL
LIN {X 0,Y 341.336,Z 715.452,A -85,B 0,C 180,E1 5202.087,E2 5202.087} C_VEL
LIN {X 0,Y 343.49,Z 720.252,A -85,B 0,C 180,E1 5200.502,E2 5200.502} C_VEL
LIN {X 0,Y 327.68,Z 895.273,A -85,B 0,C 180,E1 5197.198,E2 5197.198} C_VEL
LIN {X 0,Y 324.047,Z 917.722,A -85,B 0,C 180,E1 5196.642,E2 5196.642} C_VEL
LIN {X 0,Y 319.028,Z 940.002,A -85,B 0,C 180,E1 5195.896,E2 5195.896} C_VEL
LIN {X 0,Y 313.311,Z 959.862,A -85,B 0,C 180,E1 5195.002,E2 5195.002} C_VEL
LIN {X 0,Y 305.953,Z 980.892,A -85,B 0,C 180,E1 5193.776,E2 5193.776} C_VEL
LIN {X 0,Y 297.989,Z 1000.306,A -85,B 0,C 180,E1 5192.352,E2 5192.352} C_VEL
LIN {X 0,Y 289.121,Z 1018.796,A -85,B 0,C 180,E1 5190.632,E2 5190.632} C_VEL
LIN {X 0,Y 278.91,Z 1037.676,A -85,B 0,C 180,E1 5188.439,E2 5188.439} C_VEL
LIN {X 0,Y 268.908,Z 1054.323,A -85,B 0,C 180,E1 5186.013,E2 5186.013} C_VEL
LIN {X 0,Y 258.53,Z 1069.826,A -85,B 0,C 180,E1 5183.168,E2 5183.168} C_VEL
LIN {X 0,Y 247.727,Z 1084.813,A -85,B 0,C 180,E1 5179.715,E2 5179.715} C_VEL
LIN {X 0,Y 237.842,Z 1097.67,A -85,B 0,C 180,E1 5175.961,E2 5175.961} C_VEL
LIN {X 0,Y 228.531,Z 1109.151,A -85,B 0,C 180,E1 5171.684,E2 5171.684} C_VEL
LIN {X 0,Y 220.105,Z 1119.406,A -85,B 0,C 180,E1 5166.844,E2 5166.844} C_VEL
LIN {X 0,Y 212.867,Z 1128.185,A -85,B 0,C 180,E1 5161.425,E2 5161.425} C_VEL
LIN {X 0,Y 207.133,Z 1135.503,A -85,B 0,C 180,E1 5155.443,E2 5155.443} C_VEL
LIN {X 0,Y 203.27,Z 1141.121,A -85,B 0,C 180,E1 5149.242,E2 5149.242} C_VEL
LIN {X 0,Y 201.164,Z 1144.835,A -85,B 0,C 180,E1 5143.217,E2 5143.217} C_VEL
LIN {X 0,Y 200.264,Z 1147.185,A -85,B 0,C 180,E1 5137.17,E2 5137.17} C_VEL
LIN {X 0,Y 200.052,Z 1148.047,A -85,B 0,C 180,E1 5132.005,E2 5132.005} C_VEL
LIN {X 0,Y 200.063,Z 1147.994,A -85,B 0,C 180,E1 5127.135,E2 5127.135} C_VEL
LIN {X 0,Y 200.373,Z 1146.803,A -85,B 0,C 180,E1 5121.39,E2 5121.39} C_VEL
LIN {X 0,Y 201.434,Z 1144.299,A -85,B 0,C 180,E1 5115.63,E2 5115.63} C_VEL
LIN {X 0,Y 204.103,Z 1139.831,A -85,B 0,C 180,E1 5109.046,E2 5109.046} C_VEL
LIN {X 0,Y 208.449,Z 1133.889,A -85,B 0,C 180,E1 5102.891,E2 5102.891} C_VEL
LIN {X 0,Y 214.349,Z 1126.399,A -85,B 0,C 180,E1 5097.241,E2 5097.241} C_VEL
LIN {X 0,Y 222.369,Z 1116.694,A -85,B 0,C 180,E1 5091.647,E2 5091.647} C_VEL
LIN {X 0,Y 231.231,Z 1106.031,A -85,B 0,C 180,E1 5086.905,E2 5086.905} C_VEL
LIN {X 0,Y 240.894,Z 1093.847,A -85,B 0,C 180,E1 5082.721,E2 5082.721} C_VEL
LIN {X 0,Y 251.701,Z 1079.568,A -85,B 0,C 180,E1 5078.868,E2 5078.868} C_VEL
LIN {X 0,Y 262.267,Z 1064.637,A -85,B 0,C 180,E1 5075.683,E2 5075.683} C_VEL
LIN {X 0,Y 270.176,Z 1052.312,A -85,B 0,C 180,E1 5073.535,E2 5073.535} C_VEL
LIN {X 0,Y 254.419,Z 1058.842,A -85,B 0,C 180,E1 5070.202,E2 5070.202} C_VEL
LIN {X 0,Y 242.697,Z 1063.205,A -85,B 0,C 180,E1 5066.948,E2 5066.948} C_VEL
LIN {X 0,Y 234.296,Z 1066.199,A -85,B 0,C 180,E1 5064.042,E2 5064.042} C_VEL
LIN {X 0,Y 226.526,Z 1068.729,A -85,B 0,C 180,E1 5060.678,E2 5060.678} C_VEL
LIN {X 0,Y 220.907,Z 1070.594,A -85,B 0,C 180,E1 5057.654,E2 5057.654} C_VEL
LIN {X 0,Y 215.656,Z 1072.338,A -85,B 0,C 180,E1 5053.952,E2 5053.952} C_VEL
LIN {X 0,Y 214.951,Z 1072.56,A -85,B 0,C 180,E1 5053.324,E2 5053.324} C_VEL
LIN {X 0,Y 210.718,Z 1075.008,A -85,B 0,C 180,E1 5050.808,E2 5050.808} C_VEL
LIN {X 0,Y 203.602,Z 1079.766,A -85,B 0,C 180,E1 5046.505,E2 5046.505} C_VEL
LIN {X 0,Y 201.829,Z 1080.965,A -85,B 0,C 180,E1 5044.572,E2 5044.572} C_VEL
LIN {X 0,Y 201.987,Z 1084.401,A -85,B 0,C 180,E1 5030.887,E2 5030.887} C_VEL
LIN {X 0,Y 207.901,Z 1085.283,A -85,B 0,C 180,E1 5023.804,E2 5023.804} C_VEL
LIN {X 0,Y 214.383,Z 1085.33,A -85,B 0,C 180,E1 5019.241,E2 5019.241} C_VEL
LIN {X 0,Y 223.904,Z 1084.605,A -85,B 0,C 180,E1 5014.616,E2 5014.616} C_VEL
LIN {X 0,Y 237.207,Z 1082.536,A -85,B 0,C 180,E1 5010.174,E2 5010.174} C_VEL
LIN {X 0,Y 249.258,Z 1079.939,A -85,B 0,C 180,E1 5007.247,E2 5007.247} C_VEL
LIN {X 0,Y 238.42,Z 1094.78,A -85,B 0,C 180,E1 5003.629,E2 5003.629} C_VEL
LIN {X 0,Y 227.856,Z 1108.645,A -85,B 0,C 180,E1 4999.389,E2 4999.389} C_VEL
LIN {X 0,Y 218.527,Z 1120.497,A -85,B 0,C 180,E1 4994.799,E2 4994.799} C_VEL
LIN {X 0,Y 209.818,Z 1131.564,A -85,B 0,C 180,E1 4989.331,E2 4989.331} C_VEL
LIN {X 0,Y 202.886,Z 1140.833,A -85,B 0,C 180,E1 4983.502,E2 4983.502} C_VEL
LIN {X 0,Y 197.765,Z 1148.204,A -85,B 0,C 180,E1 4977.392,E2 4977.392} C_VEL
LIN {X 0,Y 194.281,Z 1154.3,A -85,B 0,C 180,E1 4970.8,E2 4970.8} C_VEL
LIN {X 0,Y 192.613,Z 1158.289,A -85,B 0,C 180,E1 4964.736,E2 4964.736} C_VEL
LIN {X 0,Y 192.051,Z 1161.019,A -85,B 0,C 180,E1 4958.684,E2 4958.684} C_VEL
LIN {X 0,Y 192.005,Z 1162.22,A -85,B 0,C 180,E1 4952.985,E2 4952.985} C_VEL
LIN {X 0,Y 192.029,Z 1162.317,A -85,B 0,C 180,E1 4948.21,E2 4948.21} C_VEL
LIN {X 0,Y 192.005,Z 1161.545,A -85,B 0,C 180,E1 4943.422,E2 4943.422} C_VEL
LIN {X 0,Y 192.266,Z 1159.615,A -85,B 0,C 180,E1 4937.865,E2 4937.865} C_VEL
LIN {X 0,Y 193.557,Z 1155.813,A -85,B 0,C 180,E1 4931.32,E2 4931.32} C_VEL
LIN {X 0,Y 196.22,Z 1150.714,A -85,B 0,C 180,E1 4925.094,E2 4925.094} C_VEL
LIN {X 0,Y 200.703,Z 1143.75,A -85,B 0,C 180,E1 4918.795,E2 4918.795} C_VEL
LIN {X 0,Y 206.958,Z 1135.305,A -85,B 0,C 180,E1 4912.85,E2 4912.85} C_VEL
LIN {X 0,Y 215.005,Z 1124.873,A -85,B 0,C 180,E1 4907.238,E2 4907.238} C_VEL
LIN {X 0,Y 224.758,Z 1112.493,A -85,B 0,C 180,E1 4902.019,E2 4902.019} C_VEL
LIN {X 0,Y 234.957,Z 1099.345,A -85,B 0,C 180,E1 4897.672,E2 4897.672} C_VEL
LIN {X 0,Y 245.679,Z 1084.747,A -85,B 0,C 180,E1 4893.877,E2 4893.877} C_VEL
LIN {X 0,Y 256.977,Z 1068.485,A -85,B 0,C 180,E1 4890.507,E2 4890.507} C_VEL
LIN {X 0,Y 267.381,Z 1052.206,A -85,B 0,C 180,E1 4887.825,E2 4887.825} C_VEL
LIN {X 0,Y 278.265,Z 1033.475,A -85,B 0,C 180,E1 4885.352,E2 4885.352} C_VEL
LIN {X 0,Y 288.088,Z 1014.735,A -85,B 0,C 180,E1 4883.365,E2 4883.365} C_VEL
LIN {X 0,Y 297.032,Z 995.096,A -85,B 0,C 180,E1 4881.711,E2 4881.711} C_VEL
LIN {X 0,Y 305.413,Z 974.005,A -85,B 0,C 180,E1 4880.291,E2 4880.291} C_VEL
LIN {X 0,Y 311.905,Z 954.609,A -85,B 0,C 180,E1 4879.254,E2 4879.254} C_VEL
LIN {X 0,Y 318.235,Z 931.49,A -85,B 0,C 180,E1 4878.296,E2 4878.296} C_VEL
LIN {X 0,Y 323.087,Z 908.695,A -85,B 0,C 180,E1 4877.603,E2 4877.603} C_VEL
LIN {X 0,Y 326.316,Z 885.732,A -85,B 0,C 180,E1 4877.077,E2 4877.077} C_VEL
LIN {X 0,Y 342.026,Z 722.227,A -85,B 0,C 180,E1 4873.889,E2 4873.889} C_VEL
LIN {X 0,Y 338.438,Z 715.392,A -85,B 0,C 180,E1 4871.071,E2 4871.071} C_VEL
LIN {X 0,Y 335.292,Z 709.666,A -85,B 0,C 180,E1 4867.97,E2 4867.97} C_VEL
LIN {X 0,Y 332.939,Z 705.606,A -85,B 0,C 180,E1 4864.823,E2 4864.823} C_VEL
LIN {X 0,Y 330.81,Z 702.304,A -85,B 0,C 180,E1 4859.307,E2 4859.307} C_VEL
LIN {X 0,Y 330.627,Z 702.536,A -85,B 0,C 180,E1 4856.879,E2 4856.879} C_VEL
LIN {X 0,Y 331.87,Z 705.789,A -85,B 0,C 180,E1 4851.772,E2 4851.772} C_VEL
LIN {X 0,Y 333.802,Z 710.084,A -85,B 0,C 180,E1 4848.51,E2 4848.51} C_VEL
LIN {X 0,Y 336.566,Z 715.929,A -85,B 0,C 180,E1 4845.329,E2 4845.329} C_VEL
LIN {X 0,Y 339.697,Z 722.852,A -85,B 0,C 180,E1 4842.528,E2 4842.528} C_VEL
LIN {X 0,Y 340.735,Z 725.442,A -85,B 0,C 180,E1 4841.696,E2 4841.696} C_VEL
LIN {X 0,Y 324.957,Z 895.14,A -85,B 0,C 180,E1 4838.524,E2 4838.524} C_VEL
LIN {X 0,Y 321.239,Z 917.656,A -85,B 0,C 180,E1 4837.979,E2 4837.979} C_VEL
LIN {X 0,Y 316.269,Z 939.394,A -85,B 0,C 180,E1 4837.272,E2 4837.272} C_VEL
LIN {X 0,Y 310.424,Z 959.332,A -85,B 0,C 180,E1 4836.4,E2 4836.4} C_VEL
LIN {X 0,Y 302.898,Z 980.485,A -85,B 0,C 180,E1 4835.199,E2 4835.199} C_VEL
LIN {X 0,Y 294.775,Z 999.887,A -85,B 0,C 180,E1 4833.811,E2 4833.811} C_VEL
LIN {X 0,Y 285.784,Z 1018.233,A -85,B 0,C 180,E1 4832.144,E2 4832.144} C_VEL
LIN {X 0,Y 275.352,Z 1037.106,A -85,B 0,C 180,E1 4830.002,E2 4830.002} C_VEL
LIN {X 0,Y 265.148,Z 1053.616,A -85,B 0,C 180,E1 4827.639,E2 4827.639} C_VEL
LIN {X 0,Y 254.421,Z 1069.229,A -85,B 0,C 180,E1 4824.828,E2 4824.828} C_VEL
LIN {X 0,Y 243.744,Z 1083.639,A -85,B 0,C 180,E1 4821.582,E2 4821.582} C_VEL
LIN {X 0,Y 233.324,Z 1096.631,A -85,B 0,C 180,E1 4817.847,E2 4817.847} C_VEL
LIN {X 0,Y 222.965,Z 1108.909,A -85,B 0,C 180,E1 4813.323,E2 4813.323} C_VEL
LIN {X 0,Y 214.01,Z 1119.268,A -85,B 0,C 180,E1 4808.417,E2 4808.417} C_VEL
LIN {X 0,Y 206.244,Z 1128.099,A -85,B 0,C 180,E1 4802.886,E2 4802.886} C_VEL
LIN {X 0,Y 200.015,Z 1135.515,A -85,B 0,C 180,E1 4796.737,E2 4796.737} C_VEL
LIN {X 0,Y 195.75,Z 1141.221,A -85,B 0,C 180,E1 4790.324,E2 4790.324} C_VEL
LIN {X 0,Y 193.369,Z 1144.979,A -85,B 0,C 180,E1 4784.065,E2 4784.065} C_VEL
LIN {X 0,Y 192.293,Z 1147.478,A -85,B 0,C 180,E1 4777.469,E2 4777.469} C_VEL
LIN {X 0,Y 192.058,Z 1148.338,A -85,B 0,C 180,E1 4772.088,E2 4772.088} C_VEL
LIN {X 0,Y 192.066,Z 1148.305,A -85,B 0,C 180,E1 4767.315,E2 4767.315} C_VEL
LIN {X 0,Y 192.385,Z 1147.203,A -85,B 0,C 180,E1 4761.331,E2 4761.331} C_VEL
LIN {X 0,Y 193.506,Z 1144.744,A -85,B 0,C 180,E1 4755.334,E2 4755.334} C_VEL
LIN {X 0,Y 196.178,Z 1140.613,A -85,B 0,C 180,E1 4748.785,E2 4748.785} C_VEL
LIN {X 0,Y 200.547,Z 1134.928,A -85,B 0,C 180,E1 4742.555,E2 4742.555} C_VEL
LIN {X 0,Y 206.823,Z 1127.481,A -85,B 0,C 180,E1 4736.556,E2 4736.556} C_VEL
LIN {X 0,Y 214.779,Z 1118.446,A -85,B 0,C 180,E1 4731.027,E2 4731.027} C_VEL
LIN {X 0,Y 223.828,Z 1108.014,A -85,B 0,C 180,E1 4726.18,E2 4726.18} C_VEL
LIN {X 0,Y 234.306,Z 1095.533,A -85,B 0,C 180,E1 4721.687,E2 4721.687} C_VEL
LIN {X 0,Y 244.833,Z 1082.386,A -85,B 0,C 180,E1 4717.984,E2 4717.984} C_VEL
LIN {X 0,Y 255.593,Z 1067.765,A -85,B 0,C 180,E1 4714.764,E2 4714.764} C_VEL
LIN {X 0,Y 260.721,Z 1060.283,A -85,B 0,C 180,E1 4713.351,E2 4713.351} C_VEL
LIN {X 0,Y 251.399,Z 1064.059,A -85,B 0,C 180,E1 4711.401,E2 4711.401} C_VEL
LIN {X 0,Y 238.615,Z 1068.519,A -85,B 0,C 180,E1 4707.99,E2 4707.99} C_VEL
LIN {X 0,Y 230.185,Z 1071.336,A -85,B 0,C 180,E1 4705.195,E2 4705.195} C_VEL
LIN {X 0,Y 221.423,Z 1074.089,A -85,B 0,C 180,E1 4701.455,E2 4701.455} C_VEL
LIN {X 0,Y 215.64,Z 1075.947,A -85,B 0,C 180,E1 4698.379,E2 4698.379} C_VEL
LIN {X 0,Y 210.153,Z 1077.635,A -85,B 0,C 180,E1 4694.606,E2 4694.606} C_VEL
LIN {X 0,Y 205.872,Z 1079.106,A -85,B 0,C 180,E1 4690.636,E2 4690.636} C_VEL
LIN {X 0,Y 202.655,Z 1080.495,A -85,B 0,C 180,E1 4686.232,E2 4686.232} C_VEL
LIN {X 0,Y 201.829,Z 1080.965,A -85,B 0,C 180,E1 4684.572,E2 4684.572} C_VEL
LIN {X 0,Y 199.754,Z 1082.66,A -85,B 0,C 180,E1 4682.145,E2 4682.145} C_VEL
LIN {X 0,Y 194.835,Z 1087.548,A -85,B 0,C 180,E1 4677.003,E2 4677.003} C_VEL
LIN {X 0,Y 194.385,Z 1088.615,A -85,B 0,C 180,E1 4674.75,E2 4674.75} C_VEL
LIN {X 0,Y 199.543,Z 1090.185,A -85,B 0,C 180,E1 4665.492,E2 4665.492} C_VEL
LIN {X 0,Y 208.126,Z 1090.43,A -85,B 0,C 180,E1 4658.882,E2 4658.882} C_VEL
LIN {X 0,Y 218.868,Z 1089.709,A -85,B 0,C 180,E1 4653.697,E2 4653.697} C_VEL
LIN {X 0,Y 232.492,Z 1087.72,A -85,B 0,C 180,E1 4649.219,E2 4649.219} C_VEL
LIN {X 0,Y 239.757,Z 1086.359,A -85,B 0,C 180,E1 4647.34,E2 4647.34} C_VEL
LIN {X 0,Y 228.165,Z 1101.274,A -85,B 0,C 180,E1 4643.316,E2 4643.316} C_VEL
LIN {X 0,Y 217.66,Z 1114.213,A -85,B 0,C 180,E1 4638.883,E2 4638.883} C_VEL
LIN {X 0,Y 208.025,Z 1125.685,A -85,B 0,C 180,E1 4633.799,E2 4633.799} C_VEL
LIN {X 0,Y 199.615,Z 1135.89,A -85,B 0,C 180,E1 4628.032,E2 4628.032} C_VEL
LIN {X 0,Y 193.335,Z 1143.856,A -85,B 0,C 180,E1 4622.187,E2 4622.187} C_VEL
LIN {X 0,Y 188.25,Z 1151.152,A -85,B 0,C 180,E1 4615.145,E2 4615.145} C_VEL
LIN {X 0,Y 185.579,Z 1155.974,A -85,B 0,C 180,E1 4608.861,E2 4608.861} C_VEL
LIN {X 0,Y 184.239,Z 1159.63,A -85,B 0,C 180,E1 4601.901,E2 4601.901} C_VEL
LIN {X 0,Y 184.008,Z 1161.334,A -85,B 0,C 180,E1 4596.552,E2 4596.552} C_VEL
LIN {X 0,Y 184.035,Z 1162.056,A -85,B 0,C 180,E1 4591.514,E2 4591.514} C_VEL
LIN {X 0,Y 184.007,Z 1161.875,A -85,B 0,C 180,E1 4586.261,E2 4586.261} C_VEL
LIN {X 0,Y 184.084,Z 1160.47,A -85,B 0,C 180,E1 4580.307,E2 4580.307} C_VEL
LIN {X 0,Y 184.78,Z 1157.802,A -85,B 0,C 180,E1 4574.303,E2 4574.303} C_VEL
LIN {X 0,Y 186.855,Z 1153.531,A -85,B 0,C 180,E1 4567.671,E2 4567.671} C_VEL
LIN {X 0,Y 190.852,Z 1147.223,A -85,B 0,C 180,E1 4560.842,E2 4560.842} C_VEL
LIN {X 0,Y 196.898,Z 1139.217,A -85,B 0,C 180,E1 4554.269,E2 4554.269} C_VEL
LIN {X 0,Y 204.486,Z 1129.9,A -85,B 0,C 180,E1 4548.426,E2 4548.426} C_VEL
LIN {X 0,Y 213.618,Z 1118.918,A -85,B 0,C 180,E1 4543.099,E2 4543.099} C_VEL
LIN {X 0,Y 224.139,Z 1106.22,A -85,B 0,C 180,E1 4538.268,E2 4538.268} C_VEL
LIN {X 0,Y 234.777,Z 1092.744,A -85,B 0,C 180,E1 4534.29,E2 4534.29} C_VEL
LIN {X 0,Y 247.073,Z 1076.274,A -85,B 0,C 180,E1 4530.461,E2 4530.461} C_VEL
LIN {X 0,Y 258.188,Z 1060.27,A -85,B 0,C 180,E1 4527.523,E2 4527.523} C_VEL
LIN {X 0,Y 269.148,Z 1042.766,A -85,B 0,C 180,E1 4524.982,E2 4524.982} C_VEL
LIN {X 0,Y 280.21,Z 1023.233,A -85,B 0,C 180,E1 4522.721,E2 4522.721} C_VEL
LIN {X 0,Y 290.069,Z 1003.541,A -85,B 0,C 180,E1 4520.912,E2 4520.912} C_VEL
LIN {X 0,Y 298.527,Z 983.979,A -85,B 0,C 180,E1 4519.488,E2 4519.488} C_VEL
LIN {X 0,Y 306.395,Z 962.934,A -85,B 0,C 180,E1 4518.263,E2 4518.263} C_VEL
LIN {X 0,Y 312.876,Z 941.666,A -85,B 0,C 180,E1 4517.308,E2 4517.308} C_VEL
LIN {X 0,Y 318.568,Z 918.164,A -85,B 0,C 180,E1 4516.514,E2 4516.514} C_VEL
LIN {X 0,Y 322.635,Z 895.2,A -85,B 0,C 180,E1 4515.934,E2 4515.934} C_VEL
LIN {X 0,Y 329.346,Z 829.173,A -85,B 0,C 180,E1 4514.636,E2 4514.636} C_VEL
LIN {X 0,Y 339.318,Z 727.482,A -85,B 0,C 180,E1 4512.681,E2 4512.681} C_VEL
LIN {X 0,Y 335.711,Z 720.545,A -85,B 0,C 180,E1 4509.514,E2 4509.514} C_VEL
LIN {X 0,Y 333.559,Z 716.693,A -85,B 0,C 180,E1 4507.146,E2 4507.146} C_VEL
LIN {X 0,Y 331.736,Z 713.349,A -85,B 0,C 180,E1 4504.494,E2 4504.494} C_VEL
LIN {X 0,Y 329.809,Z 710.205,A -85,B 0,C 180,E1 4499.131,E2 4499.131} C_VEL
LIN {X 0,Y 329.652,Z 710.589,A -85,B 0,C 180,E1 4496.688,E2 4496.688} C_VEL
LIN {X 0,Y 330.815,Z 713.724,A -85,B 0,C 180,E1 4491.92,E2 4491.92} C_VEL
LIN {X 0,Y 332.633,Z 717.939,A -85,B 0,C 180,E1 4488.732,E2 4488.732} C_VEL
LIN {X 0,Y 335.152,Z 723.511,A -85,B 0,C 180,E1 4485.707,E2 4485.707} C_VEL
LIN {X 0,Y 338.032,Z 730.13,A -85,B 0,C 180,E1 4483.016,E2 4483.016} C_VEL
LIN {X 0,Y 338.122,Z 730.753,A -85,B 0,C 180,E1 4482.908,E2 4482.908} C_VEL
LIN {X 0,Y 322.401,Z 895.103,A -85,B 0,C 180,E1 4479.87,E2 4479.87} C_VEL
LIN {X 0,Y 318.61,Z 917.591,A -85,B 0,C 180,E1 4479.337,E2 4479.337} C_VEL
LIN {X 0,Y 313.489,Z 939.518,A -85,B 0,C 180,E1 4478.642,E2 4478.642} C_VEL
LIN {X 0,Y 307.321,Z 960.075,A -85,B 0,C 180,E1 4477.761,E2 4477.761} C_VEL
LIN {X 0,Y 299.632,Z 981.074,A -85,B 0,C 180,E1 4476.587,E2 4476.587} C_VEL
LIN {X 0,Y 290.891,Z 1001.287,A -85,B 0,C 180,E1 4475.153,E2 4475.153} C_VEL
LIN {X 0,Y 281.578,Z 1019.705,A -85,B 0,C 180,E1 4473.487,E2 4473.487} C_VEL
LIN {X 0,Y 271.035,Z 1038.104,A -85,B 0,C 180,E1 4471.402,E2 4471.402} C_VEL
LIN {X 0,Y 260.198,Z 1055.084,A -85,B 0,C 180,E1 4468.973,E2 4468.973} C_VEL
LIN {X 0,Y 249.158,Z 1070.491,A -85,B 0,C 180,E1 4466.169,E2 4466.169} C_VEL
LIN {X 0,Y 237.267,Z 1085.766,A -85,B 0,C 180,E1 4462.639,E2 4462.639} C_VEL
LIN {X 0,Y 226.219,Z 1099.004,A -85,B 0,C 180,E1 4458.71,E2 4458.71} C_VEL
LIN {X 0,Y 216.072,Z 1110.337,A -85,B 0,C 180,E1 4454.327,E2 4454.327} C_VEL
LIN {X 0,Y 206.361,Z 1120.903,A -85,B 0,C 180,E1 4449.041,E2 4449.041} C_VEL
LIN {X 0,Y 198.387,Z 1129.576,A -85,B 0,C 180,E1 4443.323,E2 4443.323} C_VEL
LIN {X 0,Y 192.184,Z 1136.461,A -85,B 0,C 180,E1 4437.17,E2 4437.17} C_VEL
LIN {X 0,Y 187.65,Z 1142.105,A -85,B 0,C 180,E1 4430.264,E2 4430.264} C_VEL
LIN {X 0,Y 185.279,Z 1145.727,A -85,B 0,C 180,E1 4423.736,E2 4423.736} C_VEL
LIN {X 0,Y 184.273,Z 1147.895,A -85,B 0,C 180,E1 4417.169,E2 4417.169} C_VEL
LIN {X 0,Y 184.063,Z 1148.657,A -85,B 0,C 180,E1 4411.763,E2 4411.763} C_VEL
LIN {X 0,Y 184.095,Z 1148.535,A -85,B 0,C 180,E1 4406.263,E2 4406.263} C_VEL
LIN {X 0,Y 184.564,Z 1147.175,A -85,B 0,C 180,E1 4400.017,E2 4400.017} C_VEL
LIN {X 0,Y 185.961,Z 1144.586,A -85,B 0,C 180,E1 4393.764,E2 4393.764} C_VEL
LIN {X 0,Y 189.227,Z 1140.078,A -85,B 0,C 180,E1 4386.84,E2 4386.84} C_VEL
LIN {X 0,Y 194.299,Z 1134.169,A -85,B 0,C 180,E1 4380.395,E2 4380.395} C_VEL
LIN {X 0,Y 201.497,Z 1126.22,A -85,B 0,C 180,E1 4374.159,E2 4374.159} C_VEL
LIN {X 0,Y 210.214,Z 1116.809,A -85,B 0,C 180,E1 4368.613,E2 4368.613} C_VEL
LIN {X 0,Y 220.08,Z 1106.061,A -85,B 0,C 180,E1 4363.75,E2 4363.75} C_VEL
LIN {X 0,Y 230.715,Z 1093.802,A -85,B 0,C 180,E1 4359.519,E2 4359.519} C_VEL
LIN {X 0,Y 242.448,Z 1079.413,A -85,B 0,C 180,E1 4355.665,E2 4355.665} C_VEL
LIN {X 0,Y 250.96,Z 1068.161,A -85,B 0,C 180,E1 4353.232,E2 4353.232} C_VEL
LIN {X 0,Y 235.145,Z 1073.543,A -85,B 0,C 180,E1 4349.275,E2 4349.275} C_VEL
LIN {X 0,Y 225.263,Z 1076.626,A -85,B 0,C 180,E1 4346.068,E2 4346.068} C_VEL
LIN {X 0,Y 216.656,Z 1079.145,A -85,B 0,C 180,E1 4342.523,E2 4342.523} C_VEL
LIN {X 0,Y 209.824,Z 1081.127,A -85,B 0,C 180,E1 4338.908,E2 4338.908} C_VEL
LIN {X 0,Y 204.52,Z 1082.738,A -85,B 0,C 180,E1 4335.308,E2 4335.308} C_VEL
LIN {X 0,Y 200.068,Z 1084.22,A -85,B 0,C 180,E1 4331.24,E2 4331.24} C_VEL
LIN {X 0,Y 196.579,Z 1085.661,A -85,B 0,C 180,E1 4326.426,E2 4326.426} C_VEL
LIN {X 0,Y 194.39,Z 1087.281,A -85,B 0,C 180,E1 4320.001,E2 4320.001} C_VEL
LIN {X 0,Y 194.385,Z 1088.615,A -85,B 0,C 180,E1 4314.75,E2 4314.75} C_VEL
LIN {X 0,Y 194.164,Z 1089.822,A -85,B 0,C 180,E1 4312.319,E2 4312.319} C_VEL
LIN {X 0,Y 192.737,Z 1094.3,A -85,B 0,C 180,E1 4306.7,E2 4306.7} C_VEL
LIN {X 0,Y 193.985,Z 1095.127,A -85,B 0,C 180,E1 4304.457,E2 4304.457} C_VEL
LIN {X 0,Y 202.669,Z 1095.317,A -85,B 0,C 180,E1 4297.98,E2 4297.98} C_VEL
LIN {X 0,Y 213.827,Z 1094.587,A -85,B 0,C 180,E1 4292.679,E2 4292.679} C_VEL
LIN {X 0,Y 227.706,Z 1092.703,A -85,B 0,C 180,E1 4288.203,E2 4288.203} C_VEL
LIN {X 0,Y 230.271,Z 1092.402,A -85,B 0,C 180,E1 4287.459,E2 4287.459} C_VEL
LIN {X 0,Y 219.053,Z 1105.985,A -85,B 0,C 180,E1 4283.451,E2 4283.451} C_VEL
LIN {X 0,Y 208.487,Z 1118.078,A -85,B 0,C 180,E1 4278.846,E2 4278.846} C_VEL
LIN {X 0,Y 198.412,Z 1129.508,A -85,B 0,C 180,E1 4273.263,E2 4273.263} C_VEL
LIN {X 0,Y 190.511,Z 1138.536,A -85,B 0,C 180,E1 4267.503,E2 4267.503} C_VEL
LIN {X 0,Y 183.621,Z 1146.958,A -85,B 0,C 180,E1 4260.425,E2 4260.425} C_VEL
LIN {X 0,Y 179.237,Z 1153.255,A -85,B 0,C 180,E1 4253.333,E2 4253.333} C_VEL
LIN {X 0,Y 176.91,Z 1157.524,A -85,B 0,C 180,E1 4246.415,E2 4246.415} C_VEL
LIN {X 0,Y 176.088,Z 1160.31,A -85,B 0,C 180,E1 4239.808,E2 4239.808} C_VEL
LIN {X 0,Y 176.011,Z 1161.587,A -85,B 0,C 180,E1 4233.909,E2 4233.909} C_VEL
LIN {X 0,Y 176.039,Z 1161.762,A -85,B 0,C 180,E1 4228.413,E2 4228.413} C_VEL
LIN {X 0,Y 176.004,Z 1161.033,A -85,B 0,C 180,E1 4223.148,E2 4223.148} C_VEL
LIN {X 0,Y 176.292,Z 1159.32,A -85,B 0,C 180,E1 4217.554,E2 4217.554} C_VEL
LIN {X 0,Y 177.813,Z 1155.648,A -85,B 0,C 180,E1 4210.282,E2 4210.282} C_VEL
LIN {X 0,Y 180.762,Z 1150.817,A -85,B 0,C 180,E1 4203.736,E2 4203.736} C_VEL
LIN {X 0,Y 186.316,Z 1143.499,A -85,B 0,C 180,E1 4196.444,E2 4196.444} C_VEL
LIN {X 0,Y 193.457,Z 1135.105,A -85,B 0,C 180,E1 4190.143,E2 4190.143} C_VEL
LIN {X 0,Y 202.5,Z 1124.77,A -85,B 0,C 180,E1 4184.279,E2 4184.279} C_VEL
LIN {X 0,Y 212.776,Z 1113.143,A -85,B 0,C 180,E1 4179.163,E2 4179.163} C_VEL
LIN {X 0,Y 223.242,Z 1100.838,A -85,B 0,C 180,E1 4174.953,E2 4174.953} C_VEL
LIN {X 0,Y 235.418,Z 1085.774,A -85,B 0,C 180,E1 4170.915,E2 4170.915} C_VEL
LIN {X 0,Y 247.19,Z 1070.225,A -85,B 0,C 180,E1 4167.646,E2 4167.646} C_VEL
LIN {X 0,Y 258.453,Z 1053.814,A -85,B 0,C 180,E1 4164.94,E2 4164.94} C_VEL
LIN {X 0,Y 269.64,Z 1035.995,A -85,B 0,C 180,E1 4162.583,E2 4162.583} C_VEL
LIN {X 0,Y 279.493,Z 1018.362,A -85,B 0,C 180,E1 4160.721,E2 4160.721} C_VEL
LIN {X 0,Y 289.707,Z 997.653,A -85,B 0,C 180,E1 4158.976,E2 4158.976} C_VEL
LIN {X 0,Y 298.451,Z 977.197,A -85,B 0,C 180,E1 4157.613,E2 4157.613} C_VEL
LIN {X 0,Y 305.87,Z 956.256,A -85,B 0,C 180,E1 4156.522,E2 4156.522} C_VEL
LIN {X 0,Y 312.531,Z 933.386,A -85,B 0,C 180,E1 4155.601,E2 4155.601} C_VEL
LIN {X 0,Y 317.505,Z 911.329,A -85,B 0,C 180,E1 4154.948,E2 4154.948} C_VEL
LIN {X 0,Y 321.091,Z 888.129,A -85,B 0,C 180,E1 4154.425,E2 4154.425} C_VEL
LIN {X 0,Y 336.753,Z 733.046,A -85,B 0,C 180,E1 4151.474,E2 4151.474} C_VEL
LIN {X 0,Y 333.79,Z 727.187,A -85,B 0,C 180,E1 4148.613,E2 4148.613} C_VEL
LIN {X 0,Y 332.085,Z 724.038,A -85,B 0,C 180,E1 4146.569,E2 4146.569} C_VEL
LIN {X 0,Y 330.543,Z 721.094,A -85,B 0,C 180,E1 4144.163,E2 4144.163} C_VEL
LIN {X 0,Y 328.806,Z 718.11,A -85,B 0,C 180,E1 4138.954,E2 4138.954} C_VEL
LIN {X 0,Y 328.682,Z 718.65,A -85,B 0,C 180,E1 4136.511,E2 4136.511} C_VEL
LIN {X 0,Y 329.729,Z 721.541,A -85,B 0,C 180,E1 4132.157,E2 4132.157} C_VEL
LIN {X 0,Y 331.412,Z 725.645,A -85,B 0,C 180,E1 4129.043,E2 4129.043} C_VEL
LIN {X 0,Y 333.722,Z 730.99,A -85,B 0,C 180,E1 4126.132,E2 4126.132} C_VEL
LIN {X 0,Y 335.685,Z 735.788,A -85,B 0,C 180,E1 4124.142,E2 4124.142} C_VEL
LIN {X 0,Y 320.026,Z 895.043,A -85,B 0,C 180,E1 4121.238,E2 4121.238} C_VEL
LIN {X 0,Y 316.137,Z 917.653,A -85,B 0,C 180,E1 4120.715,E2 4120.715} C_VEL
LIN {X 0,Y 310.892,Z 939.641,A -85,B 0,C 180,E1 4120.036,E2 4120.036} C_VEL
LIN {X 0,Y 304.395,Z 960.816,A -85,B 0,C 180,E1 4119.15,E2 4119.15} C_VEL
LIN {X 0,Y 296.546,Z 981.659,A -85,B 0,C 180,E1 4118.005,E2 4118.005} C_VEL
LIN {X 0,Y 288.058,Z 1000.892,A -85,B 0,C 180,E1 4116.674,E2 4116.674} C_VEL
LIN {X 0,Y 278.413,Z 1019.542,A -85,B 0,C 180,E1 4115.031,E2 4115.031} C_VEL
LIN {X 0,Y 267.264,Z 1038.504,A -85,B 0,C 180,E1 4112.921,E2 4112.921} C_VEL
LIN {X 0,Y 256.116,Z 1055.456,A -85,B 0,C 180,E1 4110.526,E2 4110.526} C_VEL
LIN {X 0,Y 244.726,Z 1070.84,A -85,B 0,C 180,E1 4107.75,E2 4107.75} C_VEL
LIN {X 0,Y 232.663,Z 1085.806,A -85,B 0,C 180,E1 4104.314,E2 4104.314} C_VEL
LIN {X 0,Y 221.155,Z 1099.049,A -85,B 0,C 180,E1 4100.396,E2 4100.396} C_VEL
LIN {X 0,Y 210.292,Z 1110.65,A -85,B 0,C 180,E1 4095.886,E2 4095.886} C_VEL
LIN {X 0,Y 199.615,Z 1121.652,A -85,B 0,C 180,E1 4090.252,E2 4090.252} C_VEL
LIN {X 0,Y 191.238,Z 1130.256,A -85,B 0,C 180,E1 4084.379,E2 4084.379} C_VEL
LIN {X 0,Y 184.482,Z 1137.275,A -85,B 0,C 180,E1 4077.782,E2 4077.782} C_VEL
LIN {X 0,Y 179.705,Z 1142.793,A -85,B 0,C 180,E1 4070.519,E2 4070.519} C_VEL
LIN {X 0,Y 177.262,Z 1146.324,A -85,B 0,C 180,E1 4063.704,E2 4063.704} C_VEL
LIN {X 0,Y 176.25,Z 1148.314,A -85,B 0,C 180,E1 4056.842,E2 4056.842} C_VEL
LIN {X 0,Y 176.067,Z 1149.005,A -85,B 0,C 180,E1 4050.976,E2 4050.976} C_VEL
LIN {X 0,Y 176.151,Z 1148.66,A -85,B 0,C 180,E1 4044.789,E2 4044.789} C_VEL
LIN {X 0,Y 176.773,Z 1147.148,A -85,B 0,C 180,E1 4038.582,E2 4038.582} C_VEL
LIN {X 0,Y 178.675,Z 1144.246,A -85,B 0,C 180,E1 4031.737,E2 4031.737} C_VEL
LIN {X 0,Y 182.506,Z 1139.51,A -85,B 0,C 180,E1 4024.702,E2 4024.702} C_VEL
LIN {X 0,Y 188.777,Z 1132.772,A -85,B 0,C 180,E1 4017.659,E2 4017.659} C_VEL
LIN {X 0,Y 196.703,Z 1124.746,A -85,B 0,C 180,E1 4011.518,E2 4011.518} C_VEL
LIN {X 0,Y 206.093,Z 1115.118,A -85,B 0,C 180,E1 4006.071,E2 4006.071} C_VEL
LIN {X 0,Y 216.737,Z 1103.902,A -85,B 0,C 180,E1 4001.239,E2 4001.239} C_VEL
LIN {X 0,Y 228.093,Z 1091.364,A -85,B 0,C 180,E1 3997.078,E2 3997.078} C_VEL
LIN {X 0,Y 239.803,Z 1077.264,A -85,B 0,C 180,E1 3993.498,E2 3993.498} C_VEL
LIN {X 0,Y 241.355,Z 1075.262,A -85,B 0,C 180,E1 3993.009,E2 3993.009} C_VEL
LIN {X 0,Y 231.008,Z 1078.544,A -85,B 0,C 180,E1 3990.425,E2 3990.425} C_VEL
LIN {X 0,Y 220.816,Z 1081.576,A -85,B 0,C 180,E1 3987.216,E2 3987.216} C_VEL
LIN {X 0,Y 211.435,Z 1084.231,A -85,B 0,C 180,E1 3983.406,E2 3983.406} C_VEL
LIN {X 0,Y 204.735,Z 1086.058,A -85,B 0,C 180,E1 3979.991,E2 3979.991} C_VEL
LIN {X 0,Y 198.803,Z 1087.689,A -85,B 0,C 180,E1 3976.059,E2 3976.059} C_VEL
LIN {X 0,Y 193.9,Z 1089.169,A -85,B 0,C 180,E1 3971.602,E2 3971.602} C_VEL
LIN {X 0,Y 190.412,Z 1090.51,A -85,B 0,C 180,E1 3966.938,E2 3966.938} C_VEL
LIN {X 0,Y 188.051,Z 1092.169,A -85,B 0,C 180,E1 3960.001,E2 3960.001} C_VEL
LIN {X 0,Y 189.757,Z 1094.389,A -85,B 0,C 180,E1 3949.987,E2 3949.987} C_VEL
LIN {X 0,Y 193.985,Z 1095.127,A -85,B 0,C 180,E1 3944.457,E2 3944.457} C_VEL
LIN {X 0,Y 194.76,Z 1095.885,A -85,B 0,C 180,E1 3942.937,E2 3942.937} C_VEL
LIN {X 0,Y 194.654,Z 1099.523,A -85,B 0,C 180,E1 3939.038,E2 3939.038} C_VEL
LIN {X 0,Y 196.11,Z 1100.057,A -85,B 0,C 180,E1 3937.582,E2 3937.582} C_VEL
LIN {X 0,Y 208.013,Z 1099.409,A -85,B 0,C 180,E1 3931.898,E2 3931.898} C_VEL
LIN {X 0,Y 220.98,Z 1097.876,A -85,B 0,C 180,E1 3927.688,E2 3927.688} C_VEL
LIN {X 0,Y 209.204,Z 1111.079,A -85,B 0,C 180,E1 3923.316,E2 3923.316} C_VEL
LIN {X 0,Y 197.236,Z 1123.987,A -85,B 0,C 180,E1 3917.742,E2 3917.742} C_VEL
LIN {X 0,Y 187.517,Z 1134.425,A -85,B 0,C 180,E1 3911.799,E2 3911.799} C_VEL
LIN {X 0,Y 179.733,Z 1142.872,A -85,B 0,C 180,E1 3905.349,E2 3905.349} C_VEL
LIN {X 0,Y 173.564,Z 1150.279,A -85,B 0,C 180,E1 3897.815,E2 3897.815} C_VEL
LIN {X 0,Y 170.161,Z 1155.223,A -85,B 0,C 180,E1 3890.891,E2 3890.891} C_VEL
LIN {X 0,Y 168.359,Z 1159.017,A -85,B 0,C 180,E1 3883.106,E2 3883.106} C_VEL
LIN {X 0,Y 168.006,Z 1160.748,A -85,B 0,C 180,E1 3877.18,E2 3877.18} C_VEL
LIN {X 0,Y 168.038,Z 1161.447,A -85,B 0,C 180,E1 3872.046,E2 3872.046} C_VEL
LIN {X 0,Y 168.018,Z 1161.369,A -85,B 0,C 180,E1 3866.93,E2 3866.93} C_VEL
